NodeFactory.AddNodeAsPrototype('Vision/Basic Container Operations/F_VN_FillContainerExp/F_VN_FillContainerExp_DINT', node_F_VN_FillContainerExp_DINT);
NodeFactory.AddNodeAsPrototype('Vision/Basic Container Operations/F_VN_FillContainerExp/F_VN_FillContainerExp_INT', node_F_VN_FillContainerExp_INT);
NodeFactory.AddNodeAsPrototype('Vision/Basic Container Operations/F_VN_FillContainerExp/F_VN_FillContainerExp_ITcVnImage', node_F_VN_FillContainerExp_ITcVnImage);
NodeFactory.AddNodeAsPrototype('Vision/Basic Container Operations/F_VN_FillContainerExp/F_VN_FillContainerExp_LREAL', node_F_VN_FillContainerExp_LREAL);
NodeFactory.AddNodeAsPrototype('Vision/Basic Container Operations/F_VN_FillContainerExp/F_VN_FillContainerExp_REAL', node_F_VN_FillContainerExp_REAL);
NodeFactory.AddNodeAsPrototype('Vision/Basic Container Operations/F_VN_FillContainerExp/F_VN_FillContainerExp_SINT', node_F_VN_FillContainerExp_SINT);
NodeFactory.AddNodeAsPrototype('Vision/Basic Container Operations/F_VN_FillContainerExp/F_VN_FillContainerExp_TcVnDMatch', node_F_VN_FillContainerExp_TcVnDMatch);
NodeFactory.AddNodeAsPrototype('Vision/Basic Container Operations/F_VN_FillContainerExp/F_VN_FillContainerExp_TcVnKeyPoint', node_F_VN_FillContainerExp_TcVnKeyPoint);
NodeFactory.AddNodeAsPrototype('Vision/Basic Container Operations/F_VN_FillContainerExp/F_VN_FillContainerExp_TcVnPoint2_DINT', node_F_VN_FillContainerExp_TcVnPoint2_DINT);
NodeFactory.AddNodeAsPrototype('Vision/Basic Container Operations/F_VN_FillContainerExp/F_VN_FillContainerExp_TcVnPoint2_LREAL', node_F_VN_FillContainerExp_TcVnPoint2_LREAL);
NodeFactory.AddNodeAsPrototype('Vision/Basic Container Operations/F_VN_FillContainerExp/F_VN_FillContainerExp_TcVnPoint2_REAL', node_F_VN_FillContainerExp_TcVnPoint2_REAL);
NodeFactory.AddNodeAsPrototype('Vision/Basic Container Operations/F_VN_FillContainerExp/F_VN_FillContainerExp_TcVnPoint3_LREAL', node_F_VN_FillContainerExp_TcVnPoint3_LREAL);
NodeFactory.AddNodeAsPrototype('Vision/Basic Container Operations/F_VN_FillContainerExp/F_VN_FillContainerExp_TcVnPoint3_REAL', node_F_VN_FillContainerExp_TcVnPoint3_REAL);
NodeFactory.AddNodeAsPrototype('Vision/Basic Container Operations/F_VN_FillContainerExp/F_VN_FillContainerExp_TcVnRectangle_DINT', node_F_VN_FillContainerExp_TcVnRectangle_DINT);
NodeFactory.AddNodeAsPrototype('Vision/Basic Container Operations/F_VN_FillContainerExp/F_VN_FillContainerExp_TcVnRotatedRectangle', node_F_VN_FillContainerExp_TcVnRotatedRectangle);
NodeFactory.AddNodeAsPrototype('Vision/Basic Container Operations/F_VN_FillContainerExp/F_VN_FillContainerExp_TcVnVector2_DINT', node_F_VN_FillContainerExp_TcVnVector2_DINT);
NodeFactory.AddNodeAsPrototype('Vision/Basic Container Operations/F_VN_FillContainerExp/F_VN_FillContainerExp_TcVnVector2_INT', node_F_VN_FillContainerExp_TcVnVector2_INT);
NodeFactory.AddNodeAsPrototype('Vision/Basic Container Operations/F_VN_FillContainerExp/F_VN_FillContainerExp_TcVnVector2_REAL', node_F_VN_FillContainerExp_TcVnVector2_REAL);
NodeFactory.AddNodeAsPrototype('Vision/Basic Container Operations/F_VN_FillContainerExp/F_VN_FillContainerExp_TcVnVector2_SINT', node_F_VN_FillContainerExp_TcVnVector2_SINT);
NodeFactory.AddNodeAsPrototype('Vision/Basic Container Operations/F_VN_FillContainerExp/F_VN_FillContainerExp_TcVnVector2_UINT', node_F_VN_FillContainerExp_TcVnVector2_UINT);
NodeFactory.AddNodeAsPrototype('Vision/Basic Container Operations/F_VN_FillContainerExp/F_VN_FillContainerExp_TcVnVector2_USINT', node_F_VN_FillContainerExp_TcVnVector2_USINT);
NodeFactory.AddNodeAsPrototype('Vision/Basic Container Operations/F_VN_FillContainerExp/F_VN_FillContainerExp_TcVnVector3_INT', node_F_VN_FillContainerExp_TcVnVector3_INT);
NodeFactory.AddNodeAsPrototype('Vision/Basic Container Operations/F_VN_FillContainerExp/F_VN_FillContainerExp_TcVnVector3_REAL', node_F_VN_FillContainerExp_TcVnVector3_REAL);
NodeFactory.AddNodeAsPrototype('Vision/Basic Container Operations/F_VN_FillContainerExp/F_VN_FillContainerExp_TcVnVector3_SINT', node_F_VN_FillContainerExp_TcVnVector3_SINT);
NodeFactory.AddNodeAsPrototype('Vision/Basic Container Operations/F_VN_FillContainerExp/F_VN_FillContainerExp_TcVnVector3_UINT', node_F_VN_FillContainerExp_TcVnVector3_UINT);
NodeFactory.AddNodeAsPrototype('Vision/Basic Container Operations/F_VN_FillContainerExp/F_VN_FillContainerExp_TcVnVector3_USINT', node_F_VN_FillContainerExp_TcVnVector3_USINT);
NodeFactory.AddNodeAsPrototype('Vision/Basic Container Operations/F_VN_FillContainerExp/F_VN_FillContainerExp_TcVnVector4_DINT', node_F_VN_FillContainerExp_TcVnVector4_DINT);
NodeFactory.AddNodeAsPrototype('Vision/Basic Container Operations/F_VN_FillContainerExp/F_VN_FillContainerExp_TcVnVector4_INT', node_F_VN_FillContainerExp_TcVnVector4_INT);
NodeFactory.AddNodeAsPrototype('Vision/Basic Container Operations/F_VN_FillContainerExp/F_VN_FillContainerExp_TcVnVector4_LREAL', node_F_VN_FillContainerExp_TcVnVector4_LREAL);
NodeFactory.AddNodeAsPrototype('Vision/Basic Container Operations/F_VN_FillContainerExp/F_VN_FillContainerExp_TcVnVector4_REAL', node_F_VN_FillContainerExp_TcVnVector4_REAL);
NodeFactory.AddNodeAsPrototype('Vision/Basic Container Operations/F_VN_FillContainerExp/F_VN_FillContainerExp_TcVnVector4_SINT', node_F_VN_FillContainerExp_TcVnVector4_SINT);
NodeFactory.AddNodeAsPrototype('Vision/Basic Container Operations/F_VN_FillContainerExp/F_VN_FillContainerExp_TcVnVector4_UINT', node_F_VN_FillContainerExp_TcVnVector4_UINT);
NodeFactory.AddNodeAsPrototype('Vision/Basic Container Operations/F_VN_FillContainerExp/F_VN_FillContainerExp_TcVnVector4_USINT', node_F_VN_FillContainerExp_TcVnVector4_USINT);
NodeFactory.AddNodeAsPrototype('Vision/Basic Container Operations/F_VN_FillContainerExp/F_VN_FillContainerExp_UDINT', node_F_VN_FillContainerExp_UDINT);
NodeFactory.AddNodeAsPrototype('Vision/Basic Container Operations/F_VN_FillContainerExp/F_VN_FillContainerExp_UINT', node_F_VN_FillContainerExp_UINT);
NodeFactory.AddNodeAsPrototype('Vision/Basic Container Operations/F_VN_FillContainerExp/F_VN_FillContainerExp_ULINT', node_F_VN_FillContainerExp_ULINT);
NodeFactory.AddNodeAsPrototype('Vision/Basic Container Operations/F_VN_FillContainerExp/F_VN_FillContainerExp_USINT', node_F_VN_FillContainerExp_USINT);

NodeFactory.AddNodeAsPrototype('Vision/Basic Container Operations/F_VN_GetAt/F_VN_GetAt_DINT', node_F_VN_GetAt_DINT);
NodeFactory.AddNodeAsPrototype('Vision/Basic Container Operations/F_VN_GetAt/F_VN_GetAt_INT', node_F_VN_GetAt_INT);
NodeFactory.AddNodeAsPrototype('Vision/Basic Container Operations/F_VN_GetAt/F_VN_GetAt_ITcVnContainer', node_F_VN_GetAt_ITcVnContainer);
NodeFactory.AddNodeAsPrototype('Vision/Basic Container Operations/F_VN_GetAt/F_VN_GetAt_ITcVnImage', node_F_VN_GetAt_ITcVnImage);
NodeFactory.AddNodeAsPrototype('Vision/Basic Container Operations/F_VN_GetAt/F_VN_GetAt_LREAL', node_F_VN_GetAt_LREAL);
NodeFactory.AddNodeAsPrototype('Vision/Basic Container Operations/F_VN_GetAt/F_VN_GetAt_REAL', node_F_VN_GetAt_REAL);
NodeFactory.AddNodeAsPrototype('Vision/Basic Container Operations/F_VN_GetAt/F_VN_GetAt_SINT', node_F_VN_GetAt_SINT);
NodeFactory.AddNodeAsPrototype('Vision/Basic Container Operations/F_VN_GetAt/F_VN_GetAt_TcVnDMatch', node_F_VN_GetAt_TcVnDMatch);
NodeFactory.AddNodeAsPrototype('Vision/Basic Container Operations/F_VN_GetAt/F_VN_GetAt_TcVnKeyPoint', node_F_VN_GetAt_TcVnKeyPoint);
NodeFactory.AddNodeAsPrototype('Vision/Basic Container Operations/F_VN_GetAt/F_VN_GetAt_TcVnPoint2_DINT', node_F_VN_GetAt_TcVnPoint2_DINT);
NodeFactory.AddNodeAsPrototype('Vision/Basic Container Operations/F_VN_GetAt/F_VN_GetAt_TcVnPoint2_LREAL', node_F_VN_GetAt_TcVnPoint2_LREAL);
NodeFactory.AddNodeAsPrototype('Vision/Basic Container Operations/F_VN_GetAt/F_VN_GetAt_TcVnPoint2_REAL', node_F_VN_GetAt_TcVnPoint2_REAL);
NodeFactory.AddNodeAsPrototype('Vision/Basic Container Operations/F_VN_GetAt/F_VN_GetAt_TcVnPoint3_LREAL', node_F_VN_GetAt_TcVnPoint3_LREAL);
NodeFactory.AddNodeAsPrototype('Vision/Basic Container Operations/F_VN_GetAt/F_VN_GetAt_TcVnPoint3_REAL', node_F_VN_GetAt_TcVnPoint3_REAL);
NodeFactory.AddNodeAsPrototype('Vision/Basic Container Operations/F_VN_GetAt/F_VN_GetAt_TcVnRectangle_DINT', node_F_VN_GetAt_TcVnRectangle_DINT);
NodeFactory.AddNodeAsPrototype('Vision/Basic Container Operations/F_VN_GetAt/F_VN_GetAt_TcVnRotatedRectangle', node_F_VN_GetAt_TcVnRotatedRectangle);
NodeFactory.AddNodeAsPrototype('Vision/Basic Container Operations/F_VN_GetAt/F_VN_GetAt_TcVnVector2_DINT', node_F_VN_GetAt_TcVnVector2_DINT);
NodeFactory.AddNodeAsPrototype('Vision/Basic Container Operations/F_VN_GetAt/F_VN_GetAt_TcVnVector2_INT', node_F_VN_GetAt_TcVnVector2_INT);
NodeFactory.AddNodeAsPrototype('Vision/Basic Container Operations/F_VN_GetAt/F_VN_GetAt_TcVnVector2_REAL', node_F_VN_GetAt_TcVnVector2_REAL);
NodeFactory.AddNodeAsPrototype('Vision/Basic Container Operations/F_VN_GetAt/F_VN_GetAt_TcVnVector2_SINT', node_F_VN_GetAt_TcVnVector2_SINT);
NodeFactory.AddNodeAsPrototype('Vision/Basic Container Operations/F_VN_GetAt/F_VN_GetAt_TcVnVector2_UINT', node_F_VN_GetAt_TcVnVector2_UINT);
NodeFactory.AddNodeAsPrototype('Vision/Basic Container Operations/F_VN_GetAt/F_VN_GetAt_TcVnVector2_USINT', node_F_VN_GetAt_TcVnVector2_USINT);
NodeFactory.AddNodeAsPrototype('Vision/Basic Container Operations/F_VN_GetAt/F_VN_GetAt_TcVnVector3_INT', node_F_VN_GetAt_TcVnVector3_INT);
NodeFactory.AddNodeAsPrototype('Vision/Basic Container Operations/F_VN_GetAt/F_VN_GetAt_TcVnVector3_REAL', node_F_VN_GetAt_TcVnVector3_REAL);
NodeFactory.AddNodeAsPrototype('Vision/Basic Container Operations/F_VN_GetAt/F_VN_GetAt_TcVnVector3_SINT', node_F_VN_GetAt_TcVnVector3_SINT);
NodeFactory.AddNodeAsPrototype('Vision/Basic Container Operations/F_VN_GetAt/F_VN_GetAt_TcVnVector3_UINT', node_F_VN_GetAt_TcVnVector3_UINT);
NodeFactory.AddNodeAsPrototype('Vision/Basic Container Operations/F_VN_GetAt/F_VN_GetAt_TcVnVector3_USINT', node_F_VN_GetAt_TcVnVector3_USINT);
NodeFactory.AddNodeAsPrototype('Vision/Basic Container Operations/F_VN_GetAt/F_VN_GetAt_TcVnVector4_DINT', node_F_VN_GetAt_TcVnVector4_DINT);
NodeFactory.AddNodeAsPrototype('Vision/Basic Container Operations/F_VN_GetAt/F_VN_GetAt_TcVnVector4_INT', node_F_VN_GetAt_TcVnVector4_INT);
NodeFactory.AddNodeAsPrototype('Vision/Basic Container Operations/F_VN_GetAt/F_VN_GetAt_TcVnVector4_LREAL', node_F_VN_GetAt_TcVnVector4_LREAL);
NodeFactory.AddNodeAsPrototype('Vision/Basic Container Operations/F_VN_GetAt/F_VN_GetAt_TcVnVector4_REAL', node_F_VN_GetAt_TcVnVector4_REAL);
NodeFactory.AddNodeAsPrototype('Vision/Basic Container Operations/F_VN_GetAt/F_VN_GetAt_TcVnVector4_SINT', node_F_VN_GetAt_TcVnVector4_SINT);
NodeFactory.AddNodeAsPrototype('Vision/Basic Container Operations/F_VN_GetAt/F_VN_GetAt_TcVnVector4_UINT', node_F_VN_GetAt_TcVnVector4_UINT);
NodeFactory.AddNodeAsPrototype('Vision/Basic Container Operations/F_VN_GetAt/F_VN_GetAt_TcVnVector4_USINT', node_F_VN_GetAt_TcVnVector4_USINT);
NodeFactory.AddNodeAsPrototype('Vision/Basic Container Operations/F_VN_GetAt/F_VN_GetAt_UDINT', node_F_VN_GetAt_UDINT);
NodeFactory.AddNodeAsPrototype('Vision/Basic Container Operations/F_VN_GetAt/F_VN_GetAt_UINT', node_F_VN_GetAt_UINT);
NodeFactory.AddNodeAsPrototype('Vision/Basic Container Operations/F_VN_GetAt/F_VN_GetAt_ULINT', node_F_VN_GetAt_ULINT);
NodeFactory.AddNodeAsPrototype('Vision/Basic Container Operations/F_VN_GetAt/F_VN_GetAt_USINT', node_F_VN_GetAt_USINT);

NodeFactory.AddNodeAsPrototype('Vision/Basic Container Operations/F_VN_InsertIntoContainer/F_VN_InsertIntoContainer_DINT', node_F_VN_InsertIntoContainer_DINT);
NodeFactory.AddNodeAsPrototype('Vision/Basic Container Operations/F_VN_InsertIntoContainer/F_VN_InsertIntoContainer_INT', node_F_VN_InsertIntoContainer_INT);
NodeFactory.AddNodeAsPrototype('Vision/Basic Container Operations/F_VN_InsertIntoContainer/F_VN_InsertIntoContainer_ITcVnContainer', node_F_VN_InsertIntoContainer_ITcVnContainer);
//NodeFactory.AddNodeAsPrototype('Vision/Basic Container Operations/F_VN_InsertIntoContainer/F_VN_InsertIntoContainer_ITcVnForwardIterator', node_F_VN_InsertIntoContainer_ITcVnForwardIterator);
NodeFactory.AddNodeAsPrototype('Vision/Basic Container Operations/F_VN_InsertIntoContainer/F_VN_InsertIntoContainer_ITcVnImage', node_F_VN_InsertIntoContainer_ITcVnImage);
NodeFactory.AddNodeAsPrototype('Vision/Basic Container Operations/F_VN_InsertIntoContainer/F_VN_InsertIntoContainer_LREAL', node_F_VN_InsertIntoContainer_LREAL);
NodeFactory.AddNodeAsPrototype('Vision/Basic Container Operations/F_VN_InsertIntoContainer/F_VN_InsertIntoContainer_REAL', node_F_VN_InsertIntoContainer_REAL);
NodeFactory.AddNodeAsPrototype('Vision/Basic Container Operations/F_VN_InsertIntoContainer/F_VN_InsertIntoContainer_SINT', node_F_VN_InsertIntoContainer_SINT);
NodeFactory.AddNodeAsPrototype('Vision/Basic Container Operations/F_VN_InsertIntoContainer/F_VN_InsertIntoContainer_TcVnDMatch', node_F_VN_InsertIntoContainer_TcVnDMatch);
NodeFactory.AddNodeAsPrototype('Vision/Basic Container Operations/F_VN_InsertIntoContainer/F_VN_InsertIntoContainer_TcVnKeyPoint', node_F_VN_InsertIntoContainer_TcVnKeyPoint);
NodeFactory.AddNodeAsPrototype('Vision/Basic Container Operations/F_VN_InsertIntoContainer/F_VN_InsertIntoContainer_TcVnPoint2_DINT', node_F_VN_InsertIntoContainer_TcVnPoint2_DINT);
NodeFactory.AddNodeAsPrototype('Vision/Basic Container Operations/F_VN_InsertIntoContainer/F_VN_InsertIntoContainer_TcVnPoint2_LREAL', node_F_VN_InsertIntoContainer_TcVnPoint2_LREAL);
NodeFactory.AddNodeAsPrototype('Vision/Basic Container Operations/F_VN_InsertIntoContainer/F_VN_InsertIntoContainer_TcVnPoint2_REAL', node_F_VN_InsertIntoContainer_TcVnPoint2_REAL);
NodeFactory.AddNodeAsPrototype('Vision/Basic Container Operations/F_VN_InsertIntoContainer/F_VN_InsertIntoContainer_TcVnPoint3_LREAL', node_F_VN_InsertIntoContainer_TcVnPoint3_LREAL);
NodeFactory.AddNodeAsPrototype('Vision/Basic Container Operations/F_VN_InsertIntoContainer/F_VN_InsertIntoContainer_TcVnPoint3_REAL', node_F_VN_InsertIntoContainer_TcVnPoint3_REAL);
NodeFactory.AddNodeAsPrototype('Vision/Basic Container Operations/F_VN_InsertIntoContainer/F_VN_InsertIntoContainer_TcVnRectangle_DINT', node_F_VN_InsertIntoContainer_TcVnRectangle_DINT);
NodeFactory.AddNodeAsPrototype('Vision/Basic Container Operations/F_VN_InsertIntoContainer/F_VN_InsertIntoContainer_TcVnRotatedRectangle', node_F_VN_InsertIntoContainer_TcVnRotatedRectangle);
NodeFactory.AddNodeAsPrototype('Vision/Basic Container Operations/F_VN_InsertIntoContainer/F_VN_InsertIntoContainer_TcVnVector2_DINT', node_F_VN_InsertIntoContainer_TcVnVector2_DINT);
NodeFactory.AddNodeAsPrototype('Vision/Basic Container Operations/F_VN_InsertIntoContainer/F_VN_InsertIntoContainer_TcVnVector2_INT', node_F_VN_InsertIntoContainer_TcVnVector2_INT);
NodeFactory.AddNodeAsPrototype('Vision/Basic Container Operations/F_VN_InsertIntoContainer/F_VN_InsertIntoContainer_TcVnVector2_REAL', node_F_VN_InsertIntoContainer_TcVnVector2_REAL);
NodeFactory.AddNodeAsPrototype('Vision/Basic Container Operations/F_VN_InsertIntoContainer/F_VN_InsertIntoContainer_TcVnVector2_SINT', node_F_VN_InsertIntoContainer_TcVnVector2_SINT);
NodeFactory.AddNodeAsPrototype('Vision/Basic Container Operations/F_VN_InsertIntoContainer/F_VN_InsertIntoContainer_TcVnVector2_UINT', node_F_VN_InsertIntoContainer_TcVnVector2_UINT);
NodeFactory.AddNodeAsPrototype('Vision/Basic Container Operations/F_VN_InsertIntoContainer/F_VN_InsertIntoContainer_TcVnVector2_USINT', node_F_VN_InsertIntoContainer_TcVnVector2_USINT);
NodeFactory.AddNodeAsPrototype('Vision/Basic Container Operations/F_VN_InsertIntoContainer/F_VN_InsertIntoContainer_TcVnVector3_INT', node_F_VN_InsertIntoContainer_TcVnVector3_INT);
NodeFactory.AddNodeAsPrototype('Vision/Basic Container Operations/F_VN_InsertIntoContainer/F_VN_InsertIntoContainer_TcVnVector3_REAL', node_F_VN_InsertIntoContainer_TcVnVector3_REAL);
NodeFactory.AddNodeAsPrototype('Vision/Basic Container Operations/F_VN_InsertIntoContainer/F_VN_InsertIntoContainer_TcVnVector3_SINT', node_F_VN_InsertIntoContainer_TcVnVector3_SINT);
NodeFactory.AddNodeAsPrototype('Vision/Basic Container Operations/F_VN_InsertIntoContainer/F_VN_InsertIntoContainer_TcVnVector3_UINT', node_F_VN_InsertIntoContainer_TcVnVector3_UINT);
NodeFactory.AddNodeAsPrototype('Vision/Basic Container Operations/F_VN_InsertIntoContainer/F_VN_InsertIntoContainer_TcVnVector3_USINT', node_F_VN_InsertIntoContainer_TcVnVector3_USINT);
NodeFactory.AddNodeAsPrototype('Vision/Basic Container Operations/F_VN_InsertIntoContainer/F_VN_InsertIntoContainer_TcVnVector4_DINT', node_F_VN_InsertIntoContainer_TcVnVector4_DINT);
NodeFactory.AddNodeAsPrototype('Vision/Basic Container Operations/F_VN_InsertIntoContainer/F_VN_InsertIntoContainer_TcVnVector4_INT', node_F_VN_InsertIntoContainer_TcVnVector4_INT);
NodeFactory.AddNodeAsPrototype('Vision/Basic Container Operations/F_VN_InsertIntoContainer/F_VN_InsertIntoContainer_TcVnVector4_LREAL', node_F_VN_InsertIntoContainer_TcVnVector4_LREAL);
NodeFactory.AddNodeAsPrototype('Vision/Basic Container Operations/F_VN_InsertIntoContainer/F_VN_InsertIntoContainer_TcVnVector4_REAL', node_F_VN_InsertIntoContainer_TcVnVector4_REAL);
NodeFactory.AddNodeAsPrototype('Vision/Basic Container Operations/F_VN_InsertIntoContainer/F_VN_InsertIntoContainer_TcVnVector4_SINT', node_F_VN_InsertIntoContainer_TcVnVector4_SINT);
NodeFactory.AddNodeAsPrototype('Vision/Basic Container Operations/F_VN_InsertIntoContainer/F_VN_InsertIntoContainer_TcVnVector4_UINT', node_F_VN_InsertIntoContainer_TcVnVector4_UINT);
NodeFactory.AddNodeAsPrototype('Vision/Basic Container Operations/F_VN_InsertIntoContainer/F_VN_InsertIntoContainer_TcVnVector4_USINT', node_F_VN_InsertIntoContainer_TcVnVector4_USINT);
NodeFactory.AddNodeAsPrototype('Vision/Basic Container Operations/F_VN_InsertIntoContainer/F_VN_InsertIntoContainer_UDINT', node_F_VN_InsertIntoContainer_UDINT);
NodeFactory.AddNodeAsPrototype('Vision/Basic Container Operations/F_VN_InsertIntoContainer/F_VN_InsertIntoContainer_UINT', node_F_VN_InsertIntoContainer_UINT);
NodeFactory.AddNodeAsPrototype('Vision/Basic Container Operations/F_VN_InsertIntoContainer/F_VN_InsertIntoContainer_ULINT', node_F_VN_InsertIntoContainer_ULINT);
NodeFactory.AddNodeAsPrototype('Vision/Basic Container Operations/F_VN_InsertIntoContainer/F_VN_InsertIntoContainer_USINT', node_F_VN_InsertIntoContainer_USINT);

NodeFactory.AddNodeAsPrototype('Vision/Basic Container Operations/F_VN_SetAt/F_VN_SetAt_DINT', node_F_VN_SetAt_DINT);
NodeFactory.AddNodeAsPrototype('Vision/Basic Container Operations/F_VN_SetAt/F_VN_SetAt_INT', node_F_VN_SetAt_INT);
NodeFactory.AddNodeAsPrototype('Vision/Basic Container Operations/F_VN_SetAt/F_VN_SetAt_ITcVnContainer', node_F_VN_SetAt_ITcVnContainer);
NodeFactory.AddNodeAsPrototype('Vision/Basic Container Operations/F_VN_SetAt/F_VN_SetAt_ITcVnImage', node_F_VN_SetAt_ITcVnImage);
NodeFactory.AddNodeAsPrototype('Vision/Basic Container Operations/F_VN_SetAt/F_VN_SetAt_LREAL', node_F_VN_SetAt_LREAL);
NodeFactory.AddNodeAsPrototype('Vision/Basic Container Operations/F_VN_SetAt/F_VN_SetAt_REAL', node_F_VN_SetAt_REAL);
NodeFactory.AddNodeAsPrototype('Vision/Basic Container Operations/F_VN_SetAt/F_VN_SetAt_SINT', node_F_VN_SetAt_SINT);
NodeFactory.AddNodeAsPrototype('Vision/Basic Container Operations/F_VN_SetAt/F_VN_SetAt_TcVnDMatch', node_F_VN_SetAt_TcVnDMatch);
NodeFactory.AddNodeAsPrototype('Vision/Basic Container Operations/F_VN_SetAt/F_VN_SetAt_TcVnKeyPoint', node_F_VN_SetAt_TcVnKeyPoint);
NodeFactory.AddNodeAsPrototype('Vision/Basic Container Operations/F_VN_SetAt/F_VN_SetAt_TcVnPoint2_DINT', node_F_VN_SetAt_TcVnPoint2_DINT);
NodeFactory.AddNodeAsPrototype('Vision/Basic Container Operations/F_VN_SetAt/F_VN_SetAt_TcVnPoint2_LREAL', node_F_VN_SetAt_TcVnPoint2_LREAL);
NodeFactory.AddNodeAsPrototype('Vision/Basic Container Operations/F_VN_SetAt/F_VN_SetAt_TcVnPoint2_REAL', node_F_VN_SetAt_TcVnPoint2_REAL);
NodeFactory.AddNodeAsPrototype('Vision/Basic Container Operations/F_VN_SetAt/F_VN_SetAt_TcVnPoint3_LREAL', node_F_VN_SetAt_TcVnPoint3_LREAL);
NodeFactory.AddNodeAsPrototype('Vision/Basic Container Operations/F_VN_SetAt/F_VN_SetAt_TcVnPoint3_REAL', node_F_VN_SetAt_TcVnPoint3_REAL);
NodeFactory.AddNodeAsPrototype('Vision/Basic Container Operations/F_VN_SetAt/F_VN_SetAt_TcVnRectangle_DINT', node_F_VN_SetAt_TcVnRectangle_DINT);
NodeFactory.AddNodeAsPrototype('Vision/Basic Container Operations/F_VN_SetAt/F_VN_SetAt_TcVnRotatedRectangle', node_F_VN_SetAt_TcVnRotatedRectangle);
NodeFactory.AddNodeAsPrototype('Vision/Basic Container Operations/F_VN_SetAt/F_VN_SetAt_TcVnVector2_DINT', node_F_VN_SetAt_TcVnVector2_DINT);
NodeFactory.AddNodeAsPrototype('Vision/Basic Container Operations/F_VN_SetAt/F_VN_SetAt_TcVnVector2_INT', node_F_VN_SetAt_TcVnVector2_INT);
NodeFactory.AddNodeAsPrototype('Vision/Basic Container Operations/F_VN_SetAt/F_VN_SetAt_TcVnVector2_REAL', node_F_VN_SetAt_TcVnVector2_REAL);
NodeFactory.AddNodeAsPrototype('Vision/Basic Container Operations/F_VN_SetAt/F_VN_SetAt_TcVnVector2_SINT', node_F_VN_SetAt_TcVnVector2_SINT);
NodeFactory.AddNodeAsPrototype('Vision/Basic Container Operations/F_VN_SetAt/F_VN_SetAt_TcVnVector2_UINT', node_F_VN_SetAt_TcVnVector2_UINT);
NodeFactory.AddNodeAsPrototype('Vision/Basic Container Operations/F_VN_SetAt/F_VN_SetAt_TcVnVector2_USINT', node_F_VN_SetAt_TcVnVector2_USINT);
NodeFactory.AddNodeAsPrototype('Vision/Basic Container Operations/F_VN_SetAt/F_VN_SetAt_TcVnVector3_INT', node_F_VN_SetAt_TcVnVector3_INT);
NodeFactory.AddNodeAsPrototype('Vision/Basic Container Operations/F_VN_SetAt/F_VN_SetAt_TcVnVector3_REAL', node_F_VN_SetAt_TcVnVector3_REAL);
NodeFactory.AddNodeAsPrototype('Vision/Basic Container Operations/F_VN_SetAt/F_VN_SetAt_TcVnVector3_SINT', node_F_VN_SetAt_TcVnVector3_SINT);
NodeFactory.AddNodeAsPrototype('Vision/Basic Container Operations/F_VN_SetAt/F_VN_SetAt_TcVnVector3_UINT', node_F_VN_SetAt_TcVnVector3_UINT);
NodeFactory.AddNodeAsPrototype('Vision/Basic Container Operations/F_VN_SetAt/F_VN_SetAt_TcVnVector3_USINT', node_F_VN_SetAt_TcVnVector3_USINT);
NodeFactory.AddNodeAsPrototype('Vision/Basic Container Operations/F_VN_SetAt/F_VN_SetAt_TcVnVector4_DINT', node_F_VN_SetAt_TcVnVector4_DINT);
NodeFactory.AddNodeAsPrototype('Vision/Basic Container Operations/F_VN_SetAt/F_VN_SetAt_TcVnVector4_INT', node_F_VN_SetAt_TcVnVector4_INT);
NodeFactory.AddNodeAsPrototype('Vision/Basic Container Operations/F_VN_SetAt/F_VN_SetAt_TcVnVector4_LREAL', node_F_VN_SetAt_TcVnVector4_LREAL);
NodeFactory.AddNodeAsPrototype('Vision/Basic Container Operations/F_VN_SetAt/F_VN_SetAt_TcVnVector4_REAL', node_F_VN_SetAt_TcVnVector4_REAL);
NodeFactory.AddNodeAsPrototype('Vision/Basic Container Operations/F_VN_SetAt/F_VN_SetAt_TcVnVector4_SINT', node_F_VN_SetAt_TcVnVector4_SINT);
NodeFactory.AddNodeAsPrototype('Vision/Basic Container Operations/F_VN_SetAt/F_VN_SetAt_TcVnVector4_UINT', node_F_VN_SetAt_TcVnVector4_UINT);
NodeFactory.AddNodeAsPrototype('Vision/Basic Container Operations/F_VN_SetAt/F_VN_SetAt_TcVnVector4_USINT', node_F_VN_SetAt_TcVnVector4_USINT);
NodeFactory.AddNodeAsPrototype('Vision/Basic Container Operations/F_VN_SetAt/F_VN_SetAt_UDINT', node_F_VN_SetAt_UDINT);
NodeFactory.AddNodeAsPrototype('Vision/Basic Container Operations/F_VN_SetAt/F_VN_SetAt_UINT', node_F_VN_SetAt_UINT);
NodeFactory.AddNodeAsPrototype('Vision/Basic Container Operations/F_VN_SetAt/F_VN_SetAt_ULINT', node_F_VN_SetAt_ULINT);
NodeFactory.AddNodeAsPrototype('Vision/Basic Container Operations/F_VN_SetAt/F_VN_SetAt_USINT', node_F_VN_SetAt_USINT);

//NodeFactory.AddNodeAsPrototype('Vision/Basic Container Operations/F_VN_AdvanceIterator', node_F_VN_AdvanceIterator);
NodeFactory.AddNodeAsPrototype('Vision/Basic Container Operations/F_VN_CheckIfEmpty', node_F_VN_CheckIfEmpty);
//NodeFactory.AddNodeAsPrototype('Vision/Basic Container Operations/F_VN_CheckIfIteratorIsAtEnd', node_F_VN_CheckIfIteratorIsAtEnd);
//NodeFactory.AddNodeAsPrototype('Vision/Basic Container Operations/F_VN_ConvertContainerType', node_F_VN_ConvertContainerType);
NodeFactory.AddNodeAsPrototype('Vision/Basic Container Operations/F_VN_CopyContainer', node_F_VN_CopyContainer);
//NodeFactory.AddNodeAsPrototype('Vision/Basic Container Operations/F_VN_CopyContainerElementsConditional_ITcVnContainer', node_F_VN_CopyContainerElementsConditional_ITcVnContainer);
//NodeFactory.AddNodeAsPrototype('Vision/Basic Container Operations/F_VN_CopyContainerElementsConditional_ITcVnForwardIterator', node_F_VN_CopyContainerElementsConditional_ITcVnForwardIterator);
NodeFactory.AddNodeAsPrototype('Vision/Basic Container Operations/F_VN_CreateContainer', node_F_VN_CreateContainer);
//NodeFactory.AddNodeAsPrototype('Vision/Basic Container Operations/F_VN_CreateContainerFromArray', node_F_VN_CreateContainerFromArray);
//NodeFactory.AddNodeAsPrototype('Vision/Basic Container Operations/F_VN_EraseFromContainer', node_F_VN_EraseFromContainer);
//NodeFactory.AddNodeAsPrototype('Vision/Basic Container Operations/F_VN_ExportContainer', node_F_VN_ExportContainer);
NodeFactory.AddNodeAsPrototype('Vision/Basic Container Operations/F_VN_ExportContainer_String', node_F_VN_ExportContainer_String);
//NodeFactory.AddNodeAsPrototype('Vision/Basic Container Operations/F_VN_ExportContainerSize', node_F_VN_ExportContainerSize);
//NodeFactory.AddNodeAsPrototype('Vision/Basic Container Operations/F_VN_ExportSubContainer', node_F_VN_ExportSubContainer);
NodeFactory.AddNodeAsPrototype('Vision/Basic Container Operations/F_VN_ExportSubContainer_String', node_F_VN_ExportSubContainer_String);
//NodeFactory.AddNodeAsPrototype('Vision/Basic Container Operations/F_VN_ExportSubContainerSize', node_F_VN_ExportSubContainerSize);
NodeFactory.AddNodeAsPrototype('Vision/Basic Container Operations/F_VN_ExtractContainerRange', node_F_VN_ExtractContainerRange);
//NodeFactory.AddNodeAsPrototype('Vision/Basic Container Operations/F_VN_GetContainer', node_F_VN_GetContainer);
//NodeFactory.AddNodeAsPrototype('Vision/Basic Container Operations/F_VN_GetContainerExp', node_F_VN_GetContainerExp);
//NodeFactory.AddNodeAsPrototype('Vision/Basic Container Operations/F_VN_GetForwardIterator', node_F_VN_GetForwardIterator);
NodeFactory.AddNodeAsPrototype('Vision/Basic Container Operations/F_VN_GetNumberOfElements', node_F_VN_GetNumberOfElements);
//NodeFactory.AddNodeAsPrototype('Vision/Basic Container Operations/F_VN_GetRandomAccessIterator', node_F_VN_GetRandomAccessIterator);
//NodeFactory.AddNodeAsPrototype('Vision/Basic Container Operations/F_VN_IncrementIterator', node_F_VN_IncrementIterator);
//NodeFactory.AddNodeAsPrototype('Vision/Basic Container Operations/F_VN_IteratorDistance', node_F_VN_IteratorDistance);
//NodeFactory.AddNodeAsPrototype('Vision/Basic Container Operations/F_VN_ReserveContainerMemory', node_F_VN_ReserveContainerMemory);
NodeFactory.AddNodeAsPrototype('Vision/Basic Container Operations/F_VN_ReverseContainer', node_F_VN_ReverseContainer);
//NodeFactory.AddNodeAsPrototype('Vision/Basic Container Operations/F_VN_SetContainer', node_F_VN_SetContainer);
//NodeFactory.AddNodeAsPrototype('Vision/Basic Container Operations/F_VN_SetIteratorToBegin', node_F_VN_SetIteratorToBegin);

// Basic Image Operations
//NodeFactory.AddNodeAsPrototype('Vision/Basic Image Operations/F_VN_CombineImageChannels', node_F_VN_CombineImageChannels);
NodeFactory.AddNodeAsPrototype('Vision/Basic Image Operations/F_VN_ConvertElementType', node_F_VN_ConvertElementType);
NodeFactory.AddNodeAsPrototype('Vision/Basic Image Operations/F_VN_ConvertElementTypeExp', node_F_VN_ConvertElementTypeExp);
NodeFactory.AddNodeAsPrototype('Vision/Basic Image Operations/F_VN_CopyImage', node_F_VN_CopyImage);
NodeFactory.AddNodeAsPrototype('Vision/Basic Image Operations/F_VN_CopyImageRegion', node_F_VN_CopyImageRegion);
NodeFactory.AddNodeAsPrototype('Vision/Basic Image Operations/F_VN_CopyImageRegionToRegion', node_F_VN_CopyImageRegionToRegion);
NodeFactory.AddNodeAsPrototype('Vision/Basic Image Operations/F_VN_CopyIntoDisplayableImage', node_F_VN_CopyIntoDisplayableImage);
NodeFactory.AddNodeAsPrototype('Vision/Basic Image Operations/F_VN_CreateAssociatedImage', node_F_VN_CreateAssociatedImage);
NodeFactory.AddNodeAsPrototype('Vision/Basic Image Operations/F_VN_CreateEmptyImage', node_F_VN_CreateEmptyImage);
NodeFactory.AddNodeAsPrototype('Vision/Basic Image Operations/F_VN_CreateImage', node_F_VN_CreateImage);
NodeFactory.AddNodeAsPrototype('Vision/Basic Image Operations/F_VN_CreateImageAndSetPixels', node_F_VN_CreateImageAndSetPixels);
//NodeFactory.AddNodeAsPrototype('Vision/Basic Image Operations/F_VN_CreateImageFromArray', node_F_VN_CreateImageFromArray);
//NodeFactory.AddNodeAsPrototype('Vision/Basic Image Operations/F_VN_ExportImage', node_F_VN_ExportImage);
//NodeFactory.AddNodeAsPrototype('Vision/Basic Image Operations/F_VN_ExportImageAsBmp', node_F_VN_ExportImageAsBmp);
//NodeFactory.AddNodeAsPrototype('Vision/Basic Image Operations/F_VN_ExportImageAsBmpExp', node_F_VN_ExportImageAsBmpExp);
NodeFactory.AddNodeAsPrototype('Vision/Basic Image Operations/F_VN_ExportImageAsBmpSize', node_F_VN_ExportImageAsBmpSize);
NodeFactory.AddNodeAsPrototype('Vision/Basic Image Operations/F_VN_ExportImageAsBmpSizeExp', node_F_VN_ExportImageAsBmpSizeExp);
NodeFactory.AddNodeAsPrototype('Vision/Basic Image Operations/F_VN_ExportImageSize', node_F_VN_ExportImageSize);
NodeFactory.AddNodeAsPrototype('Vision/Basic Image Operations/F_VN_FuseImages', node_F_VN_FuseImages);
//NodeFactory.AddNodeAsPrototype('Vision/Basic Image Operations/F_VN_FuseImagesArray', node_F_VN_FuseImagesArray);
NodeFactory.AddNodeAsPrototype('Vision/Basic Image Operations/F_VN_GetImageChannel', node_F_VN_GetImageChannel);
NodeFactory.AddNodeAsPrototype('Vision/Basic Image Operations/F_VN_GetImageHeight', node_F_VN_GetImageHeight);
NodeFactory.AddNodeAsPrototype('Vision/Basic Image Operations/F_VN_GetImageInfo', node_F_VN_GetImageInfo);
NodeFactory.AddNodeAsPrototype('Vision/Basic Image Operations/F_VN_GetImageWidth', node_F_VN_GetImageWidth);
NodeFactory.AddNodeAsPrototype('Vision/Basic Image Operations/F_VN_GetPixel', node_F_VN_GetPixel);
NodeFactory.AddNodeAsPrototype('Vision/Basic Image Operations/F_VN_GetPixelFormat', node_F_VN_GetPixelFormat);
NodeFactory.AddNodeAsPrototype('Vision/Basic Image Operations/F_VN_GetRoi', node_F_VN_GetRoi);
NodeFactory.AddNodeAsPrototype('Vision/Basic Image Operations/F_VN_MixImageChannels', node_F_VN_MixImageChannels);
NodeFactory.AddNodeAsPrototype('Vision/Basic Image Operations/F_VN_ResetRoi', node_F_VN_ResetRoi);
NodeFactory.AddNodeAsPrototype('Vision/Basic Image Operations/F_VN_SetImageChannel', node_F_VN_SetImageChannel);
NodeFactory.AddNodeAsPrototype('Vision/Basic Image Operations/F_VN_SetPixel', node_F_VN_SetPixel);
NodeFactory.AddNodeAsPrototype('Vision/Basic Image Operations/F_VN_SetPixels', node_F_VN_SetPixels);
NodeFactory.AddNodeAsPrototype('Vision/Basic Image Operations/F_VN_SetPixelsExp', node_F_VN_SetPixelsExp);
NodeFactory.AddNodeAsPrototype('Vision/Basic Image Operations/F_VN_SetRoi', node_F_VN_SetRoi);
NodeFactory.AddNodeAsPrototype('Vision/Basic Image Operations/F_VN_SetRoi_TcVnRectangle_DINT', node_F_VN_SetRoi_TcVnRectangle_DINT);
NodeFactory.AddNodeAsPrototype('Vision/Basic Image Operations/F_VN_SetRoi_TcVnRectangle_UDINT', node_F_VN_SetRoi_TcVnRectangle_UDINT);
//NodeFactory.AddNodeAsPrototype('Vision/Basic Image Operations/F_VN_SplitImageChannels, node_F_VN_SplitImageChannels);
NodeFactory.AddNodeAsPrototype('Vision/Basic Image Operations/F_VN_TransformIntoDisplayableImage', node_F_VN_TransformIntoDisplayableImage); 
NodeFactory.AddNodeAsPrototype('Vision/Basic Image Operations/F_VN_TransformIntoDisplayableImageExp', node_F_VN_TransformIntoDisplayableImageExp); 
NodeFactory.AddNodeAsPrototype('Vision/Basic Image Operations/F_VN_CreateNDimensionalImage', node_F_VN_CreateNDimensionalImage);
NodeFactory.AddNodeAsPrototype('Vision/Basic Image Operations/F_VN_CreateNDimensionalImageAndSetPixels', node_F_VN_CreateNDimensionalImageAndSetPixels);
//NodeFactory.AddNodeAsPrototype('Vision/Basic Image Operations/F_VN_CreateNDimensionalImageFromArray, node_F_VN_CreateNDimensionalImageFromArray);
NodeFactory.AddNodeAsPrototype('Vision/Basic Image Operations/F_VN_GetLayoutInfo', node_F_VN_GetLayoutInfo);
NodeFactory.AddNodeAsPrototype('Vision/Basic Image Operations/F_VN_PadImageBorder', node_F_VN_PadImageBorder);
NodeFactory.AddNodeAsPrototype('Vision/Basic Image Operations/F_VN_PadImageBorderExp', node_F_VN_PadImageBorderExp);
//NodeFactory.AddNodeAsPrototype('Vision/Basic Image Operations/F_VN_ReinterpretUnsupportedImage', node_F_VN_ReinterpretUnsupportedImage);

// Code Quality
NodeFactory.AddNodeAsPrototype('Vision/Code Quality/F_VN_GradeBarcode', node_F_VN_GradeBarcode);
NodeFactory.AddNodeAsPrototype('Vision/Code Quality/F_VN_GradeBarcodeExp', node_F_VN_GradeBarcodeExp);
NodeFactory.AddNodeAsPrototype('Vision/Code Quality/F_VN_GradeDataMatrixCode', node_F_VN_GradeDataMatrixCode);
NodeFactory.AddNodeAsPrototype('Vision/Code Quality/F_VN_GradeDataMatrixCodeExp', node_F_VN_GradeDataMatrixCodeExp);
NodeFactory.AddNodeAsPrototype('Vision/Code Quality/F_VN_GradeQRCode', node_F_VN_GradeQRCode);
NodeFactory.AddNodeAsPrototype('Vision/Code Quality/F_VN_GradeQRCodeExp', node_F_VN_GradeQRCodeExp);

// Code Reading
NodeFactory.AddNodeAsPrototype('Vision/Code Reading/F_VN_AnalyzeBarcodeWalsh', node_F_VN_AnalyzeBarcodeWalsh);
NodeFactory.AddNodeAsPrototype('Vision/Code Reading/F_VN_DetectBarcodesWalsh', node_F_VN_DetectBarcodesWalsh);
NodeFactory.AddNodeAsPrototype('Vision/Code Reading/F_VN_DetectCodesNeuralNetwork', node_F_VN_DetectCodesNeuralNetwork);
NodeFactory.AddNodeAsPrototype('Vision/Code Reading/F_VN_ReadBarcode', node_F_VN_ReadBarcode);
NodeFactory.AddNodeAsPrototype('Vision/Code Reading/F_VN_ReadBarcodeExp', node_F_VN_ReadBarcodeExp);
NodeFactory.AddNodeAsPrototype('Vision/Code Reading/F_VN_ReadBarcodeExp2', node_F_VN_ReadBarcodeExp2);
NodeFactory.AddNodeAsPrototype('Vision/Code Reading/F_VN_ReadBarcodeRoi', node_F_VN_ReadBarcodeRoi);
NodeFactory.AddNodeAsPrototype('Vision/Code Reading/F_VN_ReadBarcodeRoiExp', node_F_VN_ReadBarcodeRoiExp);
NodeFactory.AddNodeAsPrototype('Vision/Code Reading/F_VN_ReadDataMatrixCode', node_F_VN_ReadDataMatrixCode);
NodeFactory.AddNodeAsPrototype('Vision/Code Reading/F_VN_ReadDataMatrixCodeExp', node_F_VN_ReadDataMatrixCodeExp);
NodeFactory.AddNodeAsPrototype('Vision/Code Reading/F_VN_ReadDataMatrixCodeExp2', node_F_VN_ReadDataMatrixCodeExp2);
NodeFactory.AddNodeAsPrototype('Vision/Code Reading/F_VN_ReadDataMatrixCodeRoi', node_F_VN_ReadDataMatrixCodeRoi);
NodeFactory.AddNodeAsPrototype('Vision/Code Reading/F_VN_ReadDataMatrixCodeRoiExp', node_F_VN_ReadDataMatrixCodeRoiExp);
NodeFactory.AddNodeAsPrototype('Vision/Code Reading/F_VN_ReadDotCodeRoi', Node_F_VN_ReadDotCodeRoi);
NodeFactory.AddNodeAsPrototype('Vision/Code Reading/F_VN_ReadDotCodeRoiExp', Node_F_VN_ReadDotCodeRoiExp);
NodeFactory.AddNodeAsPrototype('Vision/Code Reading/F_VN_ReadPharmaCode', node_F_VN_ReadPharmaCode);
NodeFactory.AddNodeAsPrototype('Vision/Code Reading/F_VN_ReadPharmaCodeExp', node_F_VN_ReadPharmaCodeExp);
NodeFactory.AddNodeAsPrototype('Vision/Code Reading/F_VN_ReadPharmaCodeExp2', node_F_VN_ReadPharmaCodeExp2);
NodeFactory.AddNodeAsPrototype('Vision/Code Reading/F_VN_ReadQRCode', node_F_VN_ReadQRCode);
NodeFactory.AddNodeAsPrototype('Vision/Code Reading/F_VN_ReadQRCodeExp', node_F_VN_ReadQRCodeExp);
NodeFactory.AddNodeAsPrototype('Vision/Code Reading/F_VN_ReadQRCodeExp2', node_F_VN_ReadQRCodeExp2);

// Constants
NodeFactory.AddNodeAsPrototype('Vision/Constants/RGBA_BLACK', node_RGBA_BLACK);
NodeFactory.AddNodeAsPrototype('Vision/Constants/RGBA_RED', node_RGBA_RED);
NodeFactory.AddNodeAsPrototype('Vision/Constants/RGBA_YELLOW', node_RGBA_YELLOW);
NodeFactory.AddNodeAsPrototype('Vision/Constants/RGBA_GREEN', node_RGBA_GREEN);
NodeFactory.AddNodeAsPrototype('Vision/Constants/RGBA_CYAN', node_RGBA_CYAN);
NodeFactory.AddNodeAsPrototype('Vision/Constants/RGBA_BLUE', node_RGBA_BLUE);
NodeFactory.AddNodeAsPrototype('Vision/Constants/RGBA_MAGENTA', node_RGBA_MAGENTA);
NodeFactory.AddNodeAsPrototype('Vision/Constants/RGBA_WHITE', node_RGBA_WHITE);
NodeFactory.AddNodeAsPrototype('Vision/Constants/RGBA_RANDOM', node_RGBA_RANDOM);
NodeFactory.AddNodeAsPrototype('Vision/Constants/ContainerType_Vector_SINT', node_ContainerType_Vector_SINT);
NodeFactory.AddNodeAsPrototype('Vision/Constants/ContainerType_Vector_USINT', node_ContainerType_Vector_USINT);
NodeFactory.AddNodeAsPrototype('Vision/Constants/ContainerType_Vector_INT', node_ContainerType_Vector_INT);
NodeFactory.AddNodeAsPrototype('Vision/Constants/ContainerType_Vector_UINT', node_ContainerType_Vector_UINT);
NodeFactory.AddNodeAsPrototype('Vision/Constants/ContainerType_Vector_DINT', node_ContainerType_Vector_DINT);
NodeFactory.AddNodeAsPrototype('Vision/Constants/ContainerType_Vector_UDINT', node_ContainerType_Vector_UDINT);
NodeFactory.AddNodeAsPrototype('Vision/Constants/ContainerType_Vector_ULINT', node_ContainerType_Vector_ULINT);
NodeFactory.AddNodeAsPrototype('Vision/Constants/ContainerType_Vector_REAL', node_ContainerType_Vector_REAL);
NodeFactory.AddNodeAsPrototype('Vision/Constants/ContainerType_Vector_LREAL', node_ContainerType_Vector_LREAL);
NodeFactory.AddNodeAsPrototype('Vision/Constants/ContainerType_Vector_ITcVnImage', node_ContainerType_Vector_ITcVnImage);
NodeFactory.AddNodeAsPrototype('Vision/Constants/ContainerType_Vector_TcVnPoint2_DINT', node_ContainerType_Vector_TcVnPoint2_DINT);
NodeFactory.AddNodeAsPrototype('Vision/Constants/ContainerType_Vector_TcVnPoint2_REAL', node_ContainerType_Vector_TcVnPoint2_REAL);
NodeFactory.AddNodeAsPrototype('Vision/Constants/ContainerType_Vector_TcVnPoint2_LREAL', node_ContainerType_Vector_TcVnPoint2_LREAL);
NodeFactory.AddNodeAsPrototype('Vision/Constants/ContainerType_Vector_TcVnPoint3_REAL', node_ContainerType_Vector_TcVnPoint3_REAL);
NodeFactory.AddNodeAsPrototype('Vision/Constants/ContainerType_Vector_TcVnPoint3_LREAL', node_ContainerType_Vector_TcVnPoint3_LREAL);
NodeFactory.AddNodeAsPrototype('Vision/Constants/ContainerType_Vector_Vector_TcVnPoint2_DINT', node_ContainerType_Vector_Vector_TcVnPoint2_DINT);
NodeFactory.AddNodeAsPrototype('Vision/Constants/ContainerType_Vector_Vector_TcVnPoint2_REAL', node_ContainerType_Vector_Vector_TcVnPoint2_REAL);
NodeFactory.AddNodeAsPrototype('Vision/Constants/ContainerType_Vector_Vector_TcVnPoint3_REAL', node_ContainerType_Vector_Vector_TcVnPoint3_REAL);
NodeFactory.AddNodeAsPrototype('Vision/Constants/ContainerType_Vector_Vector_UDINT', node_ContainerType_Vector_Vector_UDINT);
NodeFactory.AddNodeAsPrototype('Vision/Constants/ContainerType_Vector_Vector_ULINT', node_ContainerType_Vector_Vector_ULINT);
NodeFactory.AddNodeAsPrototype('Vision/Constants/ContainerType_Vector_Vector_REAL', node_ContainerType_Vector_Vector_REAL);
NodeFactory.AddNodeAsPrototype('Vision/Constants/ContainerType_Vector_Vector_LREAL', node_ContainerType_Vector_Vector_LREAL);
NodeFactory.AddNodeAsPrototype('Vision/Constants/ContainerType_Vector_TcVnVector2_SINT', node_ContainerType_Vector_TcVnVector2_SINT);
NodeFactory.AddNodeAsPrototype('Vision/Constants/ContainerType_Vector_TcVnVector2_USINT', node_ContainerType_Vector_TcVnVector2_USINT);
NodeFactory.AddNodeAsPrototype('Vision/Constants/ContainerType_Vector_TcVnVector2_INT', node_ContainerType_Vector_TcVnVector2_INT);
NodeFactory.AddNodeAsPrototype('Vision/Constants/ContainerType_Vector_TcVnVector2_UINT', node_ContainerType_Vector_TcVnVector2_UINT);
NodeFactory.AddNodeAsPrototype('Vision/Constants/ContainerType_Vector_TcVnVector2_DINT', node_ContainerType_Vector_TcVnVector2_DINT);
NodeFactory.AddNodeAsPrototype('Vision/Constants/ContainerType_Vector_TcVnVector2_REAL', node_ContainerType_Vector_TcVnVector2_REAL);
NodeFactory.AddNodeAsPrototype('Vision/Constants/ContainerType_Vector_TcVnVector3_SINT', node_ContainerType_Vector_TcVnVector3_SINT);
NodeFactory.AddNodeAsPrototype('Vision/Constants/ContainerType_Vector_TcVnVector3_USINT', node_ContainerType_Vector_TcVnVector3_USINT);
NodeFactory.AddNodeAsPrototype('Vision/Constants/ContainerType_Vector_TcVnVector3_INT', node_ContainerType_Vector_TcVnVector3_INT);
NodeFactory.AddNodeAsPrototype('Vision/Constants/ContainerType_Vector_TcVnVector3_UINT', node_ContainerType_Vector_TcVnVector3_UINT);
NodeFactory.AddNodeAsPrototype('Vision/Constants/ContainerType_Vector_TcVnVector3_REAL', node_ContainerType_Vector_TcVnVector3_REAL);
NodeFactory.AddNodeAsPrototype('Vision/Constants/ContainerType_Vector_TcVnVector4_SINT', node_ContainerType_Vector_TcVnVector4_SINT);
NodeFactory.AddNodeAsPrototype('Vision/Constants/ContainerType_Vector_TcVnVector4_USINT', node_ContainerType_Vector_TcVnVector4_USINT);
NodeFactory.AddNodeAsPrototype('Vision/Constants/ContainerType_Vector_TcVnVector4_INT', node_ContainerType_Vector_TcVnVector4_INT);
NodeFactory.AddNodeAsPrototype('Vision/Constants/ContainerType_Vector_TcVnVector4_UINT', node_ContainerType_Vector_TcVnVector4_UINT);
NodeFactory.AddNodeAsPrototype('Vision/Constants/ContainerType_Vector_TcVnVector4_DINT', node_ContainerType_Vector_TcVnVector4_DINT);
NodeFactory.AddNodeAsPrototype('Vision/Constants/ContainerType_Vector_TcVnVector4_REAL', node_ContainerType_Vector_TcVnVector4_REAL);
NodeFactory.AddNodeAsPrototype('Vision/Constants/ContainerType_Vector_TcVnVector4_LREAL', node_ContainerType_Vector_TcVnVector4_LREAL);
NodeFactory.AddNodeAsPrototype('Vision/Constants/ContainerType_Vector_TcVnRectangle_DINT', node_ContainerType_Vector_TcVnRectangle_DINT);
NodeFactory.AddNodeAsPrototype('Vision/Constants/ContainerType_Vector_TcVnRotatedRectangle', node_ContainerType_Vector_TcVnRotatedRectangle);
NodeFactory.AddNodeAsPrototype('Vision/Constants/ContainerType_Vector_TcVnKeyPoint', node_ContainerType_Vector_TcVnKeyPoint);
NodeFactory.AddNodeAsPrototype('Vision/Constants/ContainerType_Vector_TcVnDMatch', node_ContainerType_Vector_TcVnDMatch);
NodeFactory.AddNodeAsPrototype('Vision/Constants/ContainerType_Vector_Vector_TcVnDMatch', node_ContainerType_Vector_Vector_TcVnDMatch);
NodeFactory.AddNodeAsPrototype('Vision/Constants/ContainerType_String_SINT', node_ContainerType_String_SINT);
NodeFactory.AddNodeAsPrototype('Vision/Constants/ContainerType_Vector_String_SINT', node_ContainerType_Vector_String_SINT);

// Container Statistics
NodeFactory.AddNodeAsPrototype('Vision/Container Statistics/F_VN_MaxElementElementwise/F_VN_MaxElementElementwise_DINT', node_F_VN_MaxElementElementwise_DINT);
NodeFactory.AddNodeAsPrototype('Vision/Container Statistics/F_VN_MaxElementElementwise/F_VN_MaxElementElementwise_INT', node_F_VN_MaxElementElementwise_INT);
NodeFactory.AddNodeAsPrototype('Vision/Container Statistics/F_VN_MaxElementElementwise/F_VN_MaxElementElementwise_LREAL', node_F_VN_MaxElementElementwise_LREAL);
NodeFactory.AddNodeAsPrototype('Vision/Container Statistics/F_VN_MaxElementElementwise/F_VN_MaxElementElementwise_REAL', node_F_VN_MaxElementElementwise_REAL);
NodeFactory.AddNodeAsPrototype('Vision/Container Statistics/F_VN_MaxElementElementwise/F_VN_MaxElementElementwise_SINT', node_F_VN_MaxElementElementwise_SINT);
NodeFactory.AddNodeAsPrototype('Vision/Container Statistics/F_VN_MaxElementElementwise/F_VN_MaxElementElementwise_TcVnPoint2_DINT', node_F_VN_MaxElementElementwise_TcVnPoint2_DINT);
NodeFactory.AddNodeAsPrototype('Vision/Container Statistics/F_VN_MaxElementElementwise/F_VN_MaxElementElementwise_TcVnPoint2_LREAL', node_F_VN_MaxElementElementwise_TcVnPoint2_LREAL);
NodeFactory.AddNodeAsPrototype('Vision/Container Statistics/F_VN_MaxElementElementwise/F_VN_MaxElementElementwise_TcVnPoint2_REAL', node_F_VN_MaxElementElementwise_TcVnPoint2_REAL);
NodeFactory.AddNodeAsPrototype('Vision/Container Statistics/F_VN_MaxElementElementwise/F_VN_MaxElementElementwise_TcVnPoint3_LREAL', node_F_VN_MaxElementElementwise_TcVnPoint3_LREAL);
NodeFactory.AddNodeAsPrototype('Vision/Container Statistics/F_VN_MaxElementElementwise/F_VN_MaxElementElementwise_TcVnPoint3_REAL', node_F_VN_MaxElementElementwise_TcVnPoint3_REAL);
NodeFactory.AddNodeAsPrototype('Vision/Container Statistics/F_VN_MaxElementElementwise/F_VN_MaxElementElementwise_TcVnVector2_DINT', node_F_VN_MaxElementElementwise_TcVnVector2_DINT);
NodeFactory.AddNodeAsPrototype('Vision/Container Statistics/F_VN_MaxElementElementwise/F_VN_MaxElementElementwise_TcVnVector2_INT', node_F_VN_MaxElementElementwise_TcVnVector2_INT);
NodeFactory.AddNodeAsPrototype('Vision/Container Statistics/F_VN_MaxElementElementwise/F_VN_MaxElementElementwise_TcVnVector2_REAL', node_F_VN_MaxElementElementwise_TcVnVector2_REAL);
NodeFactory.AddNodeAsPrototype('Vision/Container Statistics/F_VN_MaxElementElementwise/F_VN_MaxElementElementwise_TcVnVector2_SINT', node_F_VN_MaxElementElementwise_TcVnVector2_SINT);
NodeFactory.AddNodeAsPrototype('Vision/Container Statistics/F_VN_MaxElementElementwise/F_VN_MaxElementElementwise_TcVnVector2_UINT', node_F_VN_MaxElementElementwise_TcVnVector2_UINT);
NodeFactory.AddNodeAsPrototype('Vision/Container Statistics/F_VN_MaxElementElementwise/F_VN_MaxElementElementwise_TcVnVector2_USINT', node_F_VN_MaxElementElementwise_TcVnVector2_USINT);
NodeFactory.AddNodeAsPrototype('Vision/Container Statistics/F_VN_MaxElementElementwise/F_VN_MaxElementElementwise_TcVnVector3_INT', node_F_VN_MaxElementElementwise_TcVnVector3_INT);
NodeFactory.AddNodeAsPrototype('Vision/Container Statistics/F_VN_MaxElementElementwise/F_VN_MaxElementElementwise_TcVnVector3_REAL', node_F_VN_MaxElementElementwise_TcVnVector3_REAL);
NodeFactory.AddNodeAsPrototype('Vision/Container Statistics/F_VN_MaxElementElementwise/F_VN_MaxElementElementwise_TcVnVector3_SINT', node_F_VN_MaxElementElementwise_TcVnVector3_SINT);
NodeFactory.AddNodeAsPrototype('Vision/Container Statistics/F_VN_MaxElementElementwise/F_VN_MaxElementElementwise_TcVnVector3_UINT', node_F_VN_MaxElementElementwise_TcVnVector3_UINT);
NodeFactory.AddNodeAsPrototype('Vision/Container Statistics/F_VN_MaxElementElementwise/F_VN_MaxElementElementwise_TcVnVector3_USINT', node_F_VN_MaxElementElementwise_TcVnVector3_USINT);
NodeFactory.AddNodeAsPrototype('Vision/Container Statistics/F_VN_MaxElementElementwise/F_VN_MaxElementElementwise_TcVnVector4_DINT', node_F_VN_MaxElementElementwise_TcVnVector4_DINT);
NodeFactory.AddNodeAsPrototype('Vision/Container Statistics/F_VN_MaxElementElementwise/F_VN_MaxElementElementwise_TcVnVector4_INT', node_F_VN_MaxElementElementwise_TcVnVector4_INT);
NodeFactory.AddNodeAsPrototype('Vision/Container Statistics/F_VN_MaxElementElementwise/F_VN_MaxElementElementwise_TcVnVector4_LREAL', node_F_VN_MaxElementElementwise_TcVnVector4_LREAL);
NodeFactory.AddNodeAsPrototype('Vision/Container Statistics/F_VN_MaxElementElementwise/F_VN_MaxElementElementwise_TcVnVector4_REAL', node_F_VN_MaxElementElementwise_TcVnVector4_REAL);
NodeFactory.AddNodeAsPrototype('Vision/Container Statistics/F_VN_MaxElementElementwise/F_VN_MaxElementElementwise_TcVnVector4_SINT', node_F_VN_MaxElementElementwise_TcVnVector4_SINT);
NodeFactory.AddNodeAsPrototype('Vision/Container Statistics/F_VN_MaxElementElementwise/F_VN_MaxElementElementwise_TcVnVector4_UINT', node_F_VN_MaxElementElementwise_TcVnVector4_UINT);
NodeFactory.AddNodeAsPrototype('Vision/Container Statistics/F_VN_MaxElementElementwise/F_VN_MaxElementElementwise_TcVnVector4_USINT', node_F_VN_MaxElementElementwise_TcVnVector4_USINT);
NodeFactory.AddNodeAsPrototype('Vision/Container Statistics/F_VN_MaxElementElementwise/F_VN_MaxElementElementwise_UDINT', node_F_VN_MaxElementElementwise_UDINT);
NodeFactory.AddNodeAsPrototype('Vision/Container Statistics/F_VN_MaxElementElementwise/F_VN_MaxElementElementwise_UINT', node_F_VN_MaxElementElementwise_UINT);
NodeFactory.AddNodeAsPrototype('Vision/Container Statistics/F_VN_MaxElementElementwise/F_VN_MaxElementElementwise_ULINT', node_F_VN_MaxElementElementwise_ULINT);
NodeFactory.AddNodeAsPrototype('Vision/Container Statistics/F_VN_MaxElementElementwise/F_VN_MaxElementElementwise_USINT', node_F_VN_MaxElementElementwise_USINT);

NodeFactory.AddNodeAsPrototype('Vision/Container Statistics/F_VN_MedianElementElementwise/F_VN_MedianElementElementwise_DINT', node_F_VN_MedianElementElementwise_DINT);
NodeFactory.AddNodeAsPrototype('Vision/Container Statistics/F_VN_MedianElementElementwise/F_VN_MedianElementElementwise_INT', node_F_VN_MedianElementElementwise_INT);
NodeFactory.AddNodeAsPrototype('Vision/Container Statistics/F_VN_MedianElementElementwise/F_VN_MedianElementElementwise_LREAL', node_F_VN_MedianElementElementwise_LREAL);
NodeFactory.AddNodeAsPrototype('Vision/Container Statistics/F_VN_MedianElementElementwise/F_VN_MedianElementElementwise_REAL', node_F_VN_MedianElementElementwise_REAL);
NodeFactory.AddNodeAsPrototype('Vision/Container Statistics/F_VN_MedianElementElementwise/F_VN_MedianElementElementwise_SINT', node_F_VN_MedianElementElementwise_SINT);
NodeFactory.AddNodeAsPrototype('Vision/Container Statistics/F_VN_MedianElementElementwise/F_VN_MedianElementElementwise_TcVnPoint2_DINT', node_F_VN_MedianElementElementwise_TcVnPoint2_DINT);
NodeFactory.AddNodeAsPrototype('Vision/Container Statistics/F_VN_MedianElementElementwise/F_VN_MedianElementElementwise_TcVnPoint2_LREAL', node_F_VN_MedianElementElementwise_TcVnPoint2_LREAL);
NodeFactory.AddNodeAsPrototype('Vision/Container Statistics/F_VN_MedianElementElementwise/F_VN_MedianElementElementwise_TcVnPoint2_REAL', node_F_VN_MedianElementElementwise_TcVnPoint2_REAL);
NodeFactory.AddNodeAsPrototype('Vision/Container Statistics/F_VN_MedianElementElementwise/F_VN_MedianElementElementwise_TcVnPoint3_LREAL', node_F_VN_MedianElementElementwise_TcVnPoint3_LREAL);
NodeFactory.AddNodeAsPrototype('Vision/Container Statistics/F_VN_MedianElementElementwise/F_VN_MedianElementElementwise_TcVnPoint3_REAL', node_F_VN_MedianElementElementwise_TcVnPoint3_REAL);
NodeFactory.AddNodeAsPrototype('Vision/Container Statistics/F_VN_MedianElementElementwise/F_VN_MedianElementElementwise_TcVnVector2_DINT', node_F_VN_MedianElementElementwise_TcVnVector2_DINT);
NodeFactory.AddNodeAsPrototype('Vision/Container Statistics/F_VN_MedianElementElementwise/F_VN_MedianElementElementwise_TcVnVector2_INT', node_F_VN_MedianElementElementwise_TcVnVector2_INT);
NodeFactory.AddNodeAsPrototype('Vision/Container Statistics/F_VN_MedianElementElementwise/F_VN_MedianElementElementwise_TcVnVector2_REAL', node_F_VN_MedianElementElementwise_TcVnVector2_REAL);
NodeFactory.AddNodeAsPrototype('Vision/Container Statistics/F_VN_MedianElementElementwise/F_VN_MedianElementElementwise_TcVnVector2_SINT', node_F_VN_MedianElementElementwise_TcVnVector2_SINT);
NodeFactory.AddNodeAsPrototype('Vision/Container Statistics/F_VN_MedianElementElementwise/F_VN_MedianElementElementwise_TcVnVector2_UINT', node_F_VN_MedianElementElementwise_TcVnVector2_UINT);
NodeFactory.AddNodeAsPrototype('Vision/Container Statistics/F_VN_MedianElementElementwise/F_VN_MedianElementElementwise_TcVnVector2_USINT', node_F_VN_MedianElementElementwise_TcVnVector2_USINT);
NodeFactory.AddNodeAsPrototype('Vision/Container Statistics/F_VN_MedianElementElementwise/F_VN_MedianElementElementwise_TcVnVector3_INT', node_F_VN_MedianElementElementwise_TcVnVector3_INT);
NodeFactory.AddNodeAsPrototype('Vision/Container Statistics/F_VN_MedianElementElementwise/F_VN_MedianElementElementwise_TcVnVector3_REAL', node_F_VN_MedianElementElementwise_TcVnVector3_REAL);
NodeFactory.AddNodeAsPrototype('Vision/Container Statistics/F_VN_MedianElementElementwise/F_VN_MedianElementElementwise_TcVnVector3_SINT', node_F_VN_MedianElementElementwise_TcVnVector3_SINT);
NodeFactory.AddNodeAsPrototype('Vision/Container Statistics/F_VN_MedianElementElementwise/F_VN_MedianElementElementwise_TcVnVector3_UINT', node_F_VN_MedianElementElementwise_TcVnVector3_UINT);
NodeFactory.AddNodeAsPrototype('Vision/Container Statistics/F_VN_MedianElementElementwise/F_VN_MedianElementElementwise_TcVnVector3_USINT', node_F_VN_MedianElementElementwise_TcVnVector3_USINT);
NodeFactory.AddNodeAsPrototype('Vision/Container Statistics/F_VN_MedianElementElementwise/F_VN_MedianElementElementwise_TcVnVector4_DINT', node_F_VN_MedianElementElementwise_TcVnVector4_DINT);
NodeFactory.AddNodeAsPrototype('Vision/Container Statistics/F_VN_MedianElementElementwise/F_VN_MedianElementElementwise_TcVnVector4_INT', node_F_VN_MedianElementElementwise_TcVnVector4_INT);
NodeFactory.AddNodeAsPrototype('Vision/Container Statistics/F_VN_MedianElementElementwise/F_VN_MedianElementElementwise_TcVnVector4_LREAL', node_F_VN_MedianElementElementwise_TcVnVector4_LREAL);
NodeFactory.AddNodeAsPrototype('Vision/Container Statistics/F_VN_MedianElementElementwise/F_VN_MedianElementElementwise_TcVnVector4_REAL', node_F_VN_MedianElementElementwise_TcVnVector4_REAL);
NodeFactory.AddNodeAsPrototype('Vision/Container Statistics/F_VN_MedianElementElementwise/F_VN_MedianElementElementwise_TcVnVector4_SINT', node_F_VN_MedianElementElementwise_TcVnVector4_SINT);
NodeFactory.AddNodeAsPrototype('Vision/Container Statistics/F_VN_MedianElementElementwise/F_VN_MedianElementElementwise_TcVnVector4_UINT', node_F_VN_MedianElementElementwise_TcVnVector4_UINT);
NodeFactory.AddNodeAsPrototype('Vision/Container Statistics/F_VN_MedianElementElementwise/F_VN_MedianElementElementwise_TcVnVector4_USINT', node_F_VN_MedianElementElementwise_TcVnVector4_USINT);
NodeFactory.AddNodeAsPrototype('Vision/Container Statistics/F_VN_MedianElementElementwise/F_VN_MedianElementElementwise_UDINT', node_F_VN_MedianElementElementwise_UDINT);
NodeFactory.AddNodeAsPrototype('Vision/Container Statistics/F_VN_MedianElementElementwise/F_VN_MedianElementElementwise_UINT', node_F_VN_MedianElementElementwise_UINT);
NodeFactory.AddNodeAsPrototype('Vision/Container Statistics/F_VN_MedianElementElementwise/F_VN_MedianElementElementwise_ULINT', node_F_VN_MedianElementElementwise_ULINT);
NodeFactory.AddNodeAsPrototype('Vision/Container Statistics/F_VN_MedianElementElementwise/F_VN_MedianElementElementwise_USINT', node_F_VN_MedianElementElementwise_USINT);

NodeFactory.AddNodeAsPrototype('Vision/Container Statistics/F_VN_MinElementElementwise/F_VN_MinElementElementwise_DINT', node_F_VN_MinElementElementwise_DINT);
NodeFactory.AddNodeAsPrototype('Vision/Container Statistics/F_VN_MinElementElementwise/F_VN_MinElementElementwise_INT', node_F_VN_MinElementElementwise_INT);
NodeFactory.AddNodeAsPrototype('Vision/Container Statistics/F_VN_MinElementElementwise/F_VN_MinElementElementwise_LREAL', node_F_VN_MinElementElementwise_LREAL);
NodeFactory.AddNodeAsPrototype('Vision/Container Statistics/F_VN_MinElementElementwise/F_VN_MinElementElementwise_REAL', node_F_VN_MinElementElementwise_REAL);
NodeFactory.AddNodeAsPrototype('Vision/Container Statistics/F_VN_MinElementElementwise/F_VN_MinElementElementwise_SINT', node_F_VN_MinElementElementwise_SINT);
NodeFactory.AddNodeAsPrototype('Vision/Container Statistics/F_VN_MinElementElementwise/F_VN_MinElementElementwise_TcVnPoint2_DINT', node_F_VN_MinElementElementwise_TcVnPoint2_DINT);
NodeFactory.AddNodeAsPrototype('Vision/Container Statistics/F_VN_MinElementElementwise/F_VN_MinElementElementwise_TcVnPoint2_LREAL', node_F_VN_MinElementElementwise_TcVnPoint2_LREAL);
NodeFactory.AddNodeAsPrototype('Vision/Container Statistics/F_VN_MinElementElementwise/F_VN_MinElementElementwise_TcVnPoint2_REAL', node_F_VN_MinElementElementwise_TcVnPoint2_REAL);
NodeFactory.AddNodeAsPrototype('Vision/Container Statistics/F_VN_MinElementElementwise/F_VN_MinElementElementwise_TcVnPoint3_LREAL', node_F_VN_MinElementElementwise_TcVnPoint3_LREAL);
NodeFactory.AddNodeAsPrototype('Vision/Container Statistics/F_VN_MinElementElementwise/F_VN_MinElementElementwise_TcVnPoint3_REAL', node_F_VN_MinElementElementwise_TcVnPoint3_REAL);
NodeFactory.AddNodeAsPrototype('Vision/Container Statistics/F_VN_MinElementElementwise/F_VN_MinElementElementwise_TcVnVector2_DINT', node_F_VN_MinElementElementwise_TcVnVector2_DINT);
NodeFactory.AddNodeAsPrototype('Vision/Container Statistics/F_VN_MinElementElementwise/F_VN_MinElementElementwise_TcVnVector2_INT', node_F_VN_MinElementElementwise_TcVnVector2_INT);
NodeFactory.AddNodeAsPrototype('Vision/Container Statistics/F_VN_MinElementElementwise/F_VN_MinElementElementwise_TcVnVector2_REAL', node_F_VN_MinElementElementwise_TcVnVector2_REAL);
NodeFactory.AddNodeAsPrototype('Vision/Container Statistics/F_VN_MinElementElementwise/F_VN_MinElementElementwise_TcVnVector2_SINT', node_F_VN_MinElementElementwise_TcVnVector2_SINT);
NodeFactory.AddNodeAsPrototype('Vision/Container Statistics/F_VN_MinElementElementwise/F_VN_MinElementElementwise_TcVnVector2_UINT', node_F_VN_MinElementElementwise_TcVnVector2_UINT);
NodeFactory.AddNodeAsPrototype('Vision/Container Statistics/F_VN_MinElementElementwise/F_VN_MinElementElementwise_TcVnVector2_USINT', node_F_VN_MinElementElementwise_TcVnVector2_USINT);
NodeFactory.AddNodeAsPrototype('Vision/Container Statistics/F_VN_MinElementElementwise/F_VN_MinElementElementwise_TcVnVector3_INT', node_F_VN_MinElementElementwise_TcVnVector3_INT);
NodeFactory.AddNodeAsPrototype('Vision/Container Statistics/F_VN_MinElementElementwise/F_VN_MinElementElementwise_TcVnVector3_REAL', node_F_VN_MinElementElementwise_TcVnVector3_REAL);
NodeFactory.AddNodeAsPrototype('Vision/Container Statistics/F_VN_MinElementElementwise/F_VN_MinElementElementwise_TcVnVector3_SINT', node_F_VN_MinElementElementwise_TcVnVector3_SINT);
NodeFactory.AddNodeAsPrototype('Vision/Container Statistics/F_VN_MinElementElementwise/F_VN_MinElementElementwise_TcVnVector3_UINT', node_F_VN_MinElementElementwise_TcVnVector3_UINT);
NodeFactory.AddNodeAsPrototype('Vision/Container Statistics/F_VN_MinElementElementwise/F_VN_MinElementElementwise_TcVnVector3_USINT', node_F_VN_MinElementElementwise_TcVnVector3_USINT);
NodeFactory.AddNodeAsPrototype('Vision/Container Statistics/F_VN_MinElementElementwise/F_VN_MinElementElementwise_TcVnVector4_DINT', node_F_VN_MinElementElementwise_TcVnVector4_DINT);
NodeFactory.AddNodeAsPrototype('Vision/Container Statistics/F_VN_MinElementElementwise/F_VN_MinElementElementwise_TcVnVector4_INT', node_F_VN_MinElementElementwise_TcVnVector4_INT);
NodeFactory.AddNodeAsPrototype('Vision/Container Statistics/F_VN_MinElementElementwise/F_VN_MinElementElementwise_TcVnVector4_LREAL', node_F_VN_MinElementElementwise_TcVnVector4_LREAL);
NodeFactory.AddNodeAsPrototype('Vision/Container Statistics/F_VN_MinElementElementwise/F_VN_MinElementElementwise_TcVnVector4_REAL', node_F_VN_MinElementElementwise_TcVnVector4_REAL);
NodeFactory.AddNodeAsPrototype('Vision/Container Statistics/F_VN_MinElementElementwise/F_VN_MinElementElementwise_TcVnVector4_SINT', node_F_VN_MinElementElementwise_TcVnVector4_SINT);
NodeFactory.AddNodeAsPrototype('Vision/Container Statistics/F_VN_MinElementElementwise/F_VN_MinElementElementwise_TcVnVector4_UINT', node_F_VN_MinElementElementwise_TcVnVector4_UINT);
NodeFactory.AddNodeAsPrototype('Vision/Container Statistics/F_VN_MinElementElementwise/F_VN_MinElementElementwise_TcVnVector4_USINT', node_F_VN_MinElementElementwise_TcVnVector4_USINT);
NodeFactory.AddNodeAsPrototype('Vision/Container Statistics/F_VN_MinElementElementwise/F_VN_MinElementElementwise_UDINT', node_F_VN_MinElementElementwise_UDINT);
NodeFactory.AddNodeAsPrototype('Vision/Container Statistics/F_VN_MinElementElementwise/F_VN_MinElementElementwise_UINT', node_F_VN_MinElementElementwise_UINT);
NodeFactory.AddNodeAsPrototype('Vision/Container Statistics/F_VN_MinElementElementwise/F_VN_MinElementElementwise_ULINT', node_F_VN_MinElementElementwise_ULINT);
NodeFactory.AddNodeAsPrototype('Vision/Container Statistics/F_VN_MinElementElementwise/F_VN_MinElementElementwise_USINT', node_F_VN_MinElementElementwise_USINT);
NodeFactory.AddNodeAsPrototype('Vision/Container Statistics/F_VN_ContainerAverage', node_F_VN_ContainerAverage);
NodeFactory.AddNodeAsPrototype('Vision/Container Statistics/F_VN_ContainerAverageElementwise2', node_F_VN_ContainerAverageElementwise2);
NodeFactory.AddNodeAsPrototype('Vision/Container Statistics/F_VN_ContainerAverageElementwise3', node_F_VN_ContainerAverageElementwise3);
NodeFactory.AddNodeAsPrototype('Vision/Container Statistics/F_VN_ContainerAverageElementwise4', node_F_VN_ContainerAverageElementwise4);
NodeFactory.AddNodeAsPrototype('Vision/Container Statistics/F_VN_ContainerAverageVariance', node_F_VN_ContainerAverageVariance);
NodeFactory.AddNodeAsPrototype('Vision/Container Statistics/F_VN_ContainerAverageVarianceElementwise2', node_F_VN_ContainerAverageVarianceElementwise2);
NodeFactory.AddNodeAsPrototype('Vision/Container Statistics/F_VN_ContainerAverageVarianceElementwise3', node_F_VN_ContainerAverageVarianceElementwise3);
NodeFactory.AddNodeAsPrototype('Vision/Container Statistics/F_VN_ContainerAverageVarianceElementwise4', node_F_VN_ContainerAverageVarianceElementwise4);
NodeFactory.AddNodeAsPrototype('Vision/Container Statistics/F_VN_MaxElement', node_F_VN_MaxElement);
NodeFactory.AddNodeAsPrototype('Vision/Container Statistics/F_VN_MedianElement', node_F_VN_MedianElement);
NodeFactory.AddNodeAsPrototype('Vision/Container Statistics/F_VN_MinElement', node_F_VN_MinElement);

// Contour Analysis
NodeFactory.AddNodeAsPrototype('Vision/Contour Analysis/F_VN_ApproximatePolygon', node_F_VN_ApproximatePolygon);
NodeFactory.AddNodeAsPrototype('Vision/Contour Analysis/F_VN_CheckIfPointIsInsideContour', node_F_VN_CheckIfPointIsInsideContour);
NodeFactory.AddNodeAsPrototype('Vision/Contour Analysis/F_VN_ContourArea', node_F_VN_ContourArea);
NodeFactory.AddNodeAsPrototype('Vision/Contour Analysis/F_VN_ContourCenterOfMass', node_F_VN_ContourCenterOfMass);
NodeFactory.AddNodeAsPrototype('Vision/Contour Analysis/F_VN_ContourCircularity', node_F_VN_ContourCircularity);
NodeFactory.AddNodeAsPrototype('Vision/Contour Analysis/F_VN_ContourCircularityExp', node_F_VN_ContourCircularityExp);
NodeFactory.AddNodeAsPrototype('Vision/Contour Analysis/F_VN_ContourConvexity', node_F_VN_ContourConvexity);
NodeFactory.AddNodeAsPrototype('Vision/Contour Analysis/F_VN_ContourEccentricity', node_F_VN_ContourEccentricity);
NodeFactory.AddNodeAsPrototype('Vision/Contour Analysis/F_VN_ContourElongation', node_F_VN_ContourElongation);
NodeFactory.AddNodeAsPrototype('Vision/Contour Analysis/F_VN_ContourExtremePoint', node_F_VN_ContourExtremePoint);
NodeFactory.AddNodeAsPrototype('Vision/Contour Analysis/F_VN_ContourInertiaRatio', node_F_VN_ContourInertiaRatio);
NodeFactory.AddNodeAsPrototype('Vision/Contour Analysis/F_VN_ContourMoments', node_F_VN_ContourMoments);
NodeFactory.AddNodeAsPrototype('Vision/Contour Analysis/F_VN_ContourOrientation', node_F_VN_ContourOrientation);
NodeFactory.AddNodeAsPrototype('Vision/Contour Analysis/F_VN_ContourOrientationExp', node_F_VN_ContourOrientationExp);
NodeFactory.AddNodeAsPrototype('Vision/Contour Analysis/F_VN_ContourPerimeter', node_F_VN_ContourPerimeter);
NodeFactory.AddNodeAsPrototype('Vision/Contour Analysis/F_VN_ContourRoundness', node_F_VN_ContourRoundness);
NodeFactory.AddNodeAsPrototype('Vision/Contour Analysis/F_VN_ConvexHullPoints', node_F_VN_ConvexHullPoints);
NodeFactory.AddNodeAsPrototype('Vision/Contour Analysis/F_VN_ConvexHullPointsExp', node_F_VN_ConvexHullPointsExp);
NodeFactory.AddNodeAsPrototype('Vision/Contour Analysis/F_VN_ConvexityDefects', node_F_VN_ConvexityDefects);
//NodeFactory.AddNodeAsPrototype('Vision/Contour Analysis/F_VN_CustomElementWiseContainerOperation_ITcVnContainer', node_F_VN_CustomElementWiseContainerOperation_ITcVnContainer);
//NodeFactory.AddNodeAsPrototype('Vision/Contour Analysis/F_VN_CustomElementWiseContainerOperation_ITcVnForwardIterator', node_F_VN_CustomElementWiseContainerOperation_ITcVnForwardIterator);
NodeFactory.AddNodeAsPrototype('Vision/Contour Analysis/F_VN_EnclosingCircle', node_F_VN_EnclosingCircle);
NodeFactory.AddNodeAsPrototype('Vision/Contour Analysis/F_VN_EnclosingRectangle', node_F_VN_EnclosingRectangle);
NodeFactory.AddNodeAsPrototype('Vision/Contour Analysis/F_VN_EnclosingTriangle', node_F_VN_EnclosingTriangle);
NodeFactory.AddNodeAsPrototype('Vision/Contour Analysis/F_VN_FitEllipse', node_F_VN_FitEllipse);
NodeFactory.AddNodeAsPrototype('Vision/Contour Analysis/F_VN_FitLine', node_F_VN_FitLine);
NodeFactory.AddNodeAsPrototype('Vision/Contour Analysis/F_VN_FitLineExp', node_F_VN_FitLineExp);
//NodeFactory.AddNodeAsPrototype('Vision/Contour Analysis/F_VN_FourierDescriptors', node_F_VN_FourierDescriptors);
NodeFactory.AddNodeAsPrototype('Vision/Contour Analysis/F_VN_MatchContours', node_F_VN_MatchContours);
NodeFactory.AddNodeAsPrototype('Vision/Contour Analysis/F_VN_MatchContours1vsN', node_F_VN_MatchContours1vsN);
NodeFactory.AddNodeAsPrototype('Vision/Contour Analysis/F_VN_MatchContours1vsNExp', node_F_VN_MatchContours1vsNExp);
NodeFactory.AddNodeAsPrototype('Vision/Contour Analysis/F_VN_MatchContoursExp', node_F_VN_MatchContoursExp);
NodeFactory.AddNodeAsPrototype('Vision/Contour Analysis/F_VN_UprightBoundingRectangle', node_F_VN_UprightBoundingRectangle);

// Control Functions
//NodeFactory.AddNodeAsPrototype('Vision/Control Functions/F_VN_StartAbsWatchdog', node_F_VN_StartAbsWatchdog);
//NodeFactory.AddNodeAsPrototype('Vision/Control Functions/F_VN_StartAbsWatchdogExp', node_F_VN_StartAbsWatchdogExp);
//NodeFactory.AddNodeAsPrototype('Vision/Control Functions/F_VN_StartRelWatchdog', node_F_VN_StartRelWatchdog);
//NodeFactory.AddNodeAsPrototype('Vision/Control Functions/F_VN_StartRelWatchdogExp', node_F_VN_StartRelWatchdogExp);
//NodeFactory.AddNodeAsPrototype('Vision/Control Functions/F_VN_StopWatchdog', node_F_VN_StopWatchdog);
    
// Drawing
NodeFactory.AddNodeAsPrototype('Vision/Drawing/F_VN_DrawArrow', node_F_VN_DrawArrow);
NodeFactory.AddNodeAsPrototype('Vision/Drawing/F_VN_DrawArrow_TcVnVector4_DINT', node_F_VN_DrawArrow_TcVnVector4_DINT);
NodeFactory.AddNodeAsPrototype('Vision/Drawing/F_VN_DrawArrowExp', node_F_VN_DrawArrowExp);
NodeFactory.AddNodeAsPrototype('Vision/Drawing/F_VN_DrawArrowExp_TcVnVector4_DINT', node_F_VN_DrawArrowExp_TcVnVector4_DINT);
NodeFactory.AddNodeAsPrototype('Vision/Drawing/F_VN_DrawCircle', node_F_VN_DrawCircle);
NodeFactory.AddNodeAsPrototype('Vision/Drawing/F_VN_DrawCircleExp', node_F_VN_DrawCircleExp);
NodeFactory.AddNodeAsPrototype('Vision/Drawing/F_VN_DrawCircles', node_F_VN_DrawCircles);
NodeFactory.AddNodeAsPrototype('Vision/Drawing/F_VN_DrawCirclesExp', node_F_VN_DrawCirclesExp);
NodeFactory.AddNodeAsPrototype('Vision/Drawing/F_VN_DrawCircularArc', node_F_VN_DrawCircularArc);
NodeFactory.AddNodeAsPrototype('Vision/Drawing/F_VN_DrawCircularArcExp', node_F_VN_DrawCircularArcExp);
NodeFactory.AddNodeAsPrototype('Vision/Drawing/F_VN_DrawComponents', node_F_VN_DrawComponents);
NodeFactory.AddNodeAsPrototype('Vision/Drawing/F_VN_DrawComponentsExp', node_F_VN_DrawComponentsExp);
NodeFactory.AddNodeAsPrototype('Vision/Drawing/F_VN_DrawContours', node_F_VN_DrawContours);
NodeFactory.AddNodeAsPrototype('Vision/Drawing/F_VN_DrawContoursExp', node_F_VN_DrawContoursExp);
NodeFactory.AddNodeAsPrototype('Vision/Drawing/F_VN_DrawEllipse', node_F_VN_DrawEllipse);
NodeFactory.AddNodeAsPrototype('Vision/Drawing/F_VN_DrawEllipseExp', node_F_VN_DrawEllipseExp);
NodeFactory.AddNodeAsPrototype('Vision/Drawing/F_VN_DrawKeypoints', node_F_VN_DrawKeypoints);
NodeFactory.AddNodeAsPrototype('Vision/Drawing/F_VN_DrawKeypointsExp', node_F_VN_DrawKeypointsExp);
NodeFactory.AddNodeAsPrototype('Vision/Drawing/F_VN_DrawLine', node_F_VN_DrawLine);
NodeFactory.AddNodeAsPrototype('Vision/Drawing/F_VN_DrawLine_TcVnVector4_DINT', node_F_VN_DrawLine_TcVnVector4_DINT);
NodeFactory.AddNodeAsPrototype('Vision/Drawing/F_VN_DrawLine_TcVnVector4_LREAL', node_F_VN_DrawLine_TcVnVector4_LREAL);
NodeFactory.AddNodeAsPrototype('Vision/Drawing/F_VN_DrawLineExp', node_F_VN_DrawLineExp);
NodeFactory.AddNodeAsPrototype('Vision/Drawing/F_VN_DrawLineExp_TcVnVector4_DINT', node_F_VN_DrawLineExp_TcVnVector4_DINT);
NodeFactory.AddNodeAsPrototype('Vision/Drawing/F_VN_DrawLineExp_TcVnVector4_LREAL', node_F_VN_DrawLineExp_TcVnVector4_LREAL);
NodeFactory.AddNodeAsPrototype('Vision/Drawing/F_VN_DrawLines', node_F_VN_DrawLines);
NodeFactory.AddNodeAsPrototype('Vision/Drawing/F_VN_DrawLinesExp', node_F_VN_DrawLinesExp);
NodeFactory.AddNodeAsPrototype('Vision/Drawing/F_VN_DrawMatches', node_F_VN_DrawMatches);
NodeFactory.AddNodeAsPrototype('Vision/Drawing/F_VN_DrawMatchesExp', node_F_VN_DrawMatchesExp);
NodeFactory.AddNodeAsPrototype('Vision/Drawing/F_VN_DrawOrientation', node_F_VN_DrawOrientation);
NodeFactory.AddNodeAsPrototype('Vision/Drawing/F_VN_DrawOrientationExp', node_F_VN_DrawOrientationExp);
NodeFactory.AddNodeAsPrototype('Vision/Drawing/F_VN_DrawPoint', node_F_VN_DrawPoint);
NodeFactory.AddNodeAsPrototype('Vision/Drawing/F_VN_DrawPointExp', node_F_VN_DrawPointExp);
NodeFactory.AddNodeAsPrototype('Vision/Drawing/F_VN_DrawPoints', node_F_VN_DrawPoints);
NodeFactory.AddNodeAsPrototype('Vision/Drawing/F_VN_DrawPointsExp', node_F_VN_DrawPointsExp);
NodeFactory.AddNodeAsPrototype('Vision/Drawing/F_VN_DrawPolygon', node_F_VN_DrawPolygon);
NodeFactory.AddNodeAsPrototype('Vision/Drawing/F_VN_DrawPolygonExp', node_F_VN_DrawPolygonExp);
NodeFactory.AddNodeAsPrototype('Vision/Drawing/F_VN_DrawRectangle', node_F_VN_DrawRectangle);
NodeFactory.AddNodeAsPrototype('Vision/Drawing/F_VN_DrawRectangle_TcVnRectangle_DINT', node_F_VN_DrawRectangle_TcVnRectangle_DINT);
NodeFactory.AddNodeAsPrototype('Vision/Drawing/F_VN_DrawRectangle_TcVnRectangle_UDINT', node_F_VN_DrawRectangle_TcVnRectangle_UDINT);
NodeFactory.AddNodeAsPrototype('Vision/Drawing/F_VN_DrawRotatedRectangle', node_F_VN_DrawRotatedRectangle);
NodeFactory.AddNodeAsPrototype('Vision/Drawing/F_VN_DrawRotatedRectangleExp', node_F_VN_DrawRotatedRectangleExp);
NodeFactory.AddNodeAsPrototype('Vision/Drawing/F_VN_FillCircle', node_F_VN_FillCircle);
NodeFactory.AddNodeAsPrototype('Vision/Drawing/F_VN_FillContours', node_F_VN_FillContours);
NodeFactory.AddNodeAsPrototype('Vision/Drawing/F_VN_FillEllipse', node_F_VN_FillEllipse);
NodeFactory.AddNodeAsPrototype('Vision/Drawing/F_VN_FillPolygon', node_F_VN_FillPolygon);
NodeFactory.AddNodeAsPrototype('Vision/Drawing/F_VN_FillRectangle', node_F_VN_FillRectangle);
NodeFactory.AddNodeAsPrototype('Vision/Drawing/F_VN_FillRotatedRectangle', node_F_VN_FillRotatedRectangle);
NodeFactory.AddNodeAsPrototype('Vision/Drawing/F_VN_PlotIntensityProfile', node_F_VN_PlotIntensityProfile);
NodeFactory.AddNodeAsPrototype('Vision/Drawing/F_VN_PlotIntensityProfileExp', node_F_VN_PlotIntensityProfileExp);
NodeFactory.AddNodeAsPrototype('Vision/Drawing/F_VN_PutLabel', node_F_VN_PutLabel);
NodeFactory.AddNodeAsPrototype('Vision/Drawing/F_VN_PutLabelExp', node_F_VN_PutLabelExp);
NodeFactory.AddNodeAsPrototype('Vision/Drawing/F_VN_PutText', node_F_VN_PutText);
NodeFactory.AddNodeAsPrototype('Vision/Drawing/F_VN_PutTextExp', node_F_VN_PutTextExp);

// Fourier Analysis
NodeFactory.AddNodeAsPrototype('Vision/Fourier Analysis/F_VN_CreateBandpassButterworthFilter', node_F_VN_CreateBandpassButterworthFilter);
NodeFactory.AddNodeAsPrototype('Vision/Fourier Analysis/F_VN_CreateBandpassGaussianFilter', node_F_VN_CreateBandpassGaussianFilter);
NodeFactory.AddNodeAsPrototype('Vision/Fourier Analysis/F_VN_CreateBandrejectButterworthFilter', node_F_VN_CreateBandrejectButterworthFilter);
NodeFactory.AddNodeAsPrototype('Vision/Fourier Analysis/F_VN_CreateBandrejectGaussianFilter', node_F_VN_CreateBandrejectGaussianFilter);
NodeFactory.AddNodeAsPrototype('Vision/Fourier Analysis/F_VN_CreateHighpassButterworthFilter', node_F_VN_CreateHighpassButterworthFilter);
NodeFactory.AddNodeAsPrototype('Vision/Fourier Analysis/F_VN_CreateHighpassGaussianFilter', node_F_VN_CreateHighpassGaussianFilter);
NodeFactory.AddNodeAsPrototype('Vision/Fourier Analysis/F_VN_CreateLowpassButterworthFilter', node_F_VN_CreateLowpassButterworthFilter);
NodeFactory.AddNodeAsPrototype('Vision/Fourier Analysis/F_VN_CreateLowpassGaussianFilter', node_F_VN_CreateLowpassGaussianFilter);
NodeFactory.AddNodeAsPrototype('Vision/Fourier Analysis/F_VN_Dft', node_F_VN_Dft);
NodeFactory.AddNodeAsPrototype('Vision/Fourier Analysis/F_VN_InverseDft', node_F_VN_InverseDft);
NodeFactory.AddNodeAsPrototype('Vision/Fourier Analysis/F_VN_OptimalDftSize', node_F_VN_OptimalDftSize);

// Geometric and Coordinate Transformations
NodeFactory.AddNodeAsPrototype('Vision/Geometric and Coordinate Transformations/Calibration/F_VN_CalibrateCamera', node_F_VN_CalibrateCamera);
//NodeFactory.AddNodeAsPrototype('Vision/Geometric and Coordinate Transformations/Calibration/F_VN_CalibrateCameraExp', node_F_VN_CalibrateCameraExp);
//NodeFactory.AddNodeAsPrototype('Vision/Geometric and Coordinate Transformations/Calibration/F_VN_CalibrateCameraExp2', node_F_VN_CalibrateCameraExp2);
//NodeFactory.AddNodeAsPrototype('Vision/Geometric and Coordinate Transformations/Calibration/F_VN_CalibrateCameraExp3', node_F_VN_CalibrateCameraExp3);
NodeFactory.AddNodeAsPrototype('Vision/Geometric and Coordinate Transformations/Calibration/F_VN_CalibrateCameraManually', node_F_VN_CalibrateCameraManually);
NodeFactory.AddNodeAsPrototype('Vision/Geometric and Coordinate Transformations/Calibration/F_VN_CalibrateCameraManuallyExp', node_F_VN_CalibrateCameraManuallyExp);
NodeFactory.AddNodeAsPrototype('Vision/Geometric and Coordinate Transformations/Calibration/F_VN_CalibrateCameraPlanar', node_F_VN_CalibrateCameraPlanar);
NodeFactory.AddNodeAsPrototype('Vision/Geometric and Coordinate Transformations/Calibration/F_VN_CalibrateCameraPlanarExp', node_F_VN_CalibrateCameraPlanarExp);
//NodeFactory.AddNodeAsPrototype('Vision/Geometric and Coordinate Transformations/Calibration/F_VN_CalibrateLinescanCamera', node_F_VN_CalibrateLinescanCamera);
//NodeFactory.AddNodeAsPrototype('Vision/Geometric and Coordinate Transformations/Calibration/F_VN_CalibrateLinescanCameraExp', node_F_VN_CalibrateLinescanCameraExp);
NodeFactory.AddNodeAsPrototype('Vision/Geometric and Coordinate Transformations/Calibration/F_VN_CompensateLensDistortion', node_F_VN_CompensateLensDistortion);
NodeFactory.AddNodeAsPrototype('Vision/Geometric and Coordinate Transformations/Calibration/F_VN_CompensateLensDistortionExp1', node_F_VN_CompensateLensDistortionExp1);
NodeFactory.AddNodeAsPrototype('Vision/Geometric and Coordinate Transformations/Calibration/F_VN_CompensateLensDistortionExp2', node_F_VN_CompensateLensDistortionExp2);
NodeFactory.AddNodeAsPrototype('Vision/Geometric and Coordinate Transformations/Calibration/F_VN_CompensateLensDistortionForPoints', node_F_VN_CompensateLensDistortionForPoints);
NodeFactory.AddNodeAsPrototype('Vision/Geometric and Coordinate Transformations/Calibration/F_VN_CompensateLensDistortionForPointsExp1', node_F_VN_CompensateLensDistortionForPointsExp1);
NodeFactory.AddNodeAsPrototype('Vision/Geometric and Coordinate Transformations/Calibration/F_VN_CompensateLensDistortionForPointsExp2', node_F_VN_CompensateLensDistortionForPointsExp2);
NodeFactory.AddNodeAsPrototype('Vision/Geometric and Coordinate Transformations/Calibration/F_VN_DetectPatternPoints', node_F_VN_DetectPatternPoints);
NodeFactory.AddNodeAsPrototype('Vision/Geometric and Coordinate Transformations/Calibration/F_VN_DetectPatternPointsExp', node_F_VN_DetectPatternPointsExp);
NodeFactory.AddNodeAsPrototype('Vision/Geometric and Coordinate Transformations/Calibration/F_VN_DetectPatternPoints2', node_F_VN_DetectPatternPoints2);
NodeFactory.AddNodeAsPrototype('Vision/Geometric and Coordinate Transformations/Calibration/F_VN_GenerateCalibrationPatternReferencePoints', node_F_VN_GenerateCalibrationPatternReferencePoints);
NodeFactory.AddNodeAsPrototype('Vision/Geometric and Coordinate Transformations/Calibration/F_VN_ImagePointsWorldDistance', node_F_VN_ImagePointsWorldDistance);
NodeFactory.AddNodeAsPrototype('Vision/Geometric and Coordinate Transformations/Calibration/F_VN_SolvePnP', node_F_VN_SolvePnP);
NodeFactory.AddNodeAsPrototype('Vision/Geometric and Coordinate Transformations/Calibration/F_VN_SolvePnPExp', node_F_VN_SolvePnPExp);
NodeFactory.AddNodeAsPrototype('Vision/Geometric and Coordinate Transformations/Calibration/F_VN_SortAxisAlignedPatternPoints', node_F_VN_SortAxisAlignedPatternPoints);
NodeFactory.AddNodeAsPrototype('Vision/Geometric and Coordinate Transformations/Calibration/F_VN_SortDetectedPatternPoints', node_F_VN_SortDetectedPatternPoints);
NodeFactory.AddNodeAsPrototype('Vision/Geometric and Coordinate Transformations/Calibration/F_VN_TransformCoordinatesImageToWorld_Container', node_F_VN_TransformCoordinatesImageToWorld_Container);
NodeFactory.AddNodeAsPrototype('Vision/Geometric and Coordinate Transformations/Calibration/F_VN_TransformCoordinatesImageToWorld_Point', node_F_VN_TransformCoordinatesImageToWorld_Point);
NodeFactory.AddNodeAsPrototype('Vision/Geometric and Coordinate Transformations/Calibration/F_VN_TransformCoordinatesPlanar_Container', node_F_VN_TransformCoordinatesPlanar_Container);
NodeFactory.AddNodeAsPrototype('Vision/Geometric and Coordinate Transformations/Calibration/F_VN_TransformCoordinatesPlanar_Point', node_F_VN_TransformCoordinatesPlanar_Point);
NodeFactory.AddNodeAsPrototype('Vision/Geometric and Coordinate Transformations/Calibration/F_VN_TransformCoordinatesWorldToImage_Container', node_F_VN_TransformCoordinatesWorldToImage_Container);
NodeFactory.AddNodeAsPrototype('Vision/Geometric and Coordinate Transformations/Calibration/F_VN_TransformCoordinatesWorldToImage_Point', node_F_VN_TransformCoordinatesWorldToImage_Point);
NodeFactory.AddNodeAsPrototype('Vision/Geometric and Coordinate Transformations/F_VN_AlignRotatedImageRegion', node_F_VN_AlignRotatedImageRegion);
NodeFactory.AddNodeAsPrototype('Vision/Geometric and Coordinate Transformations/F_VN_AlignRotatedImageRegionExp', node_F_VN_AlignRotatedImageRegionExp);
NodeFactory.AddNodeAsPrototype('Vision/Geometric and Coordinate Transformations/F_VN_ApplyRotationToAffineTransformation', node_F_VN_ApplyRotationToAffineTransformation);
NodeFactory.AddNodeAsPrototype('Vision/Geometric and Coordinate Transformations/F_VN_ApplyRotationToAffineTransformationExp', node_F_VN_ApplyRotationToAffineTransformationExp);
NodeFactory.AddNodeAsPrototype('Vision/Geometric and Coordinate Transformations/F_VN_ApplyScalingToAffineTransformation', node_F_VN_ApplyScalingToAffineTransformation);
NodeFactory.AddNodeAsPrototype('Vision/Geometric and Coordinate Transformations/F_VN_ApplyScalingToAffineTransformationExp', node_F_VN_ApplyScalingToAffineTransformationExp);
NodeFactory.AddNodeAsPrototype('Vision/Geometric and Coordinate Transformations/F_VN_ApplyTranslationToAffineTransformation', node_F_VN_ApplyTranslationToAffineTransformation);
NodeFactory.AddNodeAsPrototype('Vision/Geometric and Coordinate Transformations/F_VN_ApplyTranslationToAffineTransformationExp', node_F_VN_ApplyTranslationToAffineTransformationExp);
NodeFactory.AddNodeAsPrototype('Vision/Geometric and Coordinate Transformations/F_VN_ApplyYAxisInversionToAffineTransformation', node_F_VN_ApplyYAxisInversionToAffineTransformation);
NodeFactory.AddNodeAsPrototype('Vision/Geometric and Coordinate Transformations/F_VN_ApplyYAxisInversionToAffineTransformationExp', node_F_VN_ApplyYAxisInversionToAffineTransformationExp);
NodeFactory.AddNodeAsPrototype('Vision/Polarization/F_VN_DemosaicPolarizedImage', node_F_VN_DemosaicPolarizedImage);
NodeFactory.AddNodeAsPrototype('Vision/Polarization/F_VN_AngleAndDegreeOfLinearPolarization', node_F_VN_AngleAndDegreeOfLinearPolarization);
NodeFactory.AddNodeAsPrototype('Vision/Polarization/F_VN_PolarizedImageGlareReduction', node_F_VN_PolarizedImageGlareReduction);
NodeFactory.AddNodeAsPrototype('Vision/Geometric and Coordinate Transformations/F_VN_ConvertCartesianToPolarAngleImage', node_F_VN_ConvertCartesianToPolarAngleImage);
NodeFactory.AddNodeAsPrototype('Vision/Geometric and Coordinate Transformations/F_VN_ConvertCartesianToPolarAngleImageExp', node_F_VN_ConvertCartesianToPolarAngleImageExp);
NodeFactory.AddNodeAsPrototype('Vision/Geometric and Coordinate Transformations/F_VN_ConvertCartesianToPolarAngles', node_F_VN_ConvertCartesianToPolarAngles);
NodeFactory.AddNodeAsPrototype('Vision/Geometric and Coordinate Transformations/F_VN_ConvertCartesianToPolarAnglesExp', node_F_VN_ConvertCartesianToPolarAnglesExp);
NodeFactory.AddNodeAsPrototype('Vision/Geometric and Coordinate Transformations/F_VN_ConvertCartesianToPolarImages', node_F_VN_ConvertCartesianToPolarImages);
NodeFactory.AddNodeAsPrototype('Vision/Geometric and Coordinate Transformations/F_VN_ConvertCartesianToPolarImagesExp', node_F_VN_ConvertCartesianToPolarImagesExp);
NodeFactory.AddNodeAsPrototype('Vision/Geometric and Coordinate Transformations/F_VN_ConvertCartesianToPolarMagnitudeImage', node_F_VN_ConvertCartesianToPolarMagnitudeImage);
NodeFactory.AddNodeAsPrototype('Vision/Geometric and Coordinate Transformations/F_VN_ConvertCartesianToPolarMagnitudes', node_F_VN_ConvertCartesianToPolarMagnitudes);
NodeFactory.AddNodeAsPrototype('Vision/Geometric and Coordinate Transformations/F_VN_ConvertCartesianToPolarPoints', node_F_VN_ConvertCartesianToPolarPoints);
NodeFactory.AddNodeAsPrototype('Vision/Geometric and Coordinate Transformations/F_VN_ConvertCartesianToPolarPointsExp', node_F_VN_ConvertCartesianToPolarPointsExp);
NodeFactory.AddNodeAsPrototype('Vision/Geometric and Coordinate Transformations/F_VN_ConvertPolarToCartesianImages', node_F_VN_ConvertPolarToCartesianImages);
NodeFactory.AddNodeAsPrototype('Vision/Geometric and Coordinate Transformations/F_VN_ConvertPolarToCartesianImagesExp', node_F_VN_ConvertPolarToCartesianImagesExp);
NodeFactory.AddNodeAsPrototype('Vision/Geometric and Coordinate Transformations/F_VN_ConvertPolarToCartesianPoints', node_F_VN_ConvertPolarToCartesianPoints);
NodeFactory.AddNodeAsPrototype('Vision/Geometric and Coordinate Transformations/F_VN_ConvertPolarToCartesianPointsExp', node_F_VN_ConvertPolarToCartesianPointsExp);
NodeFactory.AddNodeAsPrototype('Vision/Geometric and Coordinate Transformations/F_VN_DecomposeAffineTransformation', node_F_VN_DecomposeAffineTransformation);
NodeFactory.AddNodeAsPrototype('Vision/Geometric and Coordinate Transformations/F_VN_DecomposeAffineTransformationExp', node_F_VN_DecomposeAffineTransformationExp);
NodeFactory.AddNodeAsPrototype('Vision/Geometric and Coordinate Transformations/F_VN_DecomposeHomography', node_F_VN_DecomposeHomography);
NodeFactory.AddNodeAsPrototype('Vision/Geometric and Coordinate Transformations/F_VN_DecomposeHomographyExp', node_F_VN_DecomposeHomographyExp);
NodeFactory.AddNodeAsPrototype('Vision/Geometric and Coordinate Transformations/F_VN_FlipImage', node_F_VN_FlipImage);
NodeFactory.AddNodeAsPrototype('Vision/Geometric and Coordinate Transformations/F_VN_GenerateAffineTransformationUnitMatrix2D', node_F_VN_GenerateAffineTransformationUnitMatrix2D);
NodeFactory.AddNodeAsPrototype('Vision/Geometric and Coordinate Transformations/F_VN_GetAffineTransformation', node_F_VN_GetAffineTransformation);
NodeFactory.AddNodeAsPrototype('Vision/Geometric and Coordinate Transformations/F_VN_GetAffineTransformation2D', node_F_VN_GetAffineTransformation2D);
//NodeFactory.AddNodeAsPrototype('Vision/Geometric and Coordinate Transformations/F_VN_GetAffineTransformation2DExp', node_F_VN_GetAffineTransformation2DExp);
NodeFactory.AddNodeAsPrototype('Vision/Geometric and Coordinate Transformations/F_VN_GetPerspectiveTransformation', node_F_VN_GetPerspectiveTransformation);
NodeFactory.AddNodeAsPrototype('Vision/Geometric and Coordinate Transformations/F_VN_Homography', node_F_VN_Homography);
NodeFactory.AddNodeAsPrototype('Vision/Geometric and Coordinate Transformations/F_VN_HomographyExp', node_F_VN_HomographyExp);
NodeFactory.AddNodeAsPrototype('Vision/Geometric and Coordinate Transformations/F_VN_InvertAffineTransformation', node_F_VN_InvertAffineTransformation);
NodeFactory.AddNodeAsPrototype('Vision/Geometric and Coordinate Transformations/F_VN_PerspectiveTransformation', node_F_VN_PerspectiveTransformation);
NodeFactory.AddNodeAsPrototype('Vision/Geometric and Coordinate Transformations/F_VN_PyramidDown', node_F_VN_PyramidDown);
NodeFactory.AddNodeAsPrototype('Vision/Geometric and Coordinate Transformations/F_VN_PyramidUp', node_F_VN_PyramidUp);
NodeFactory.AddNodeAsPrototype('Vision/Geometric and Coordinate Transformations/F_VN_ConvertMaps', node_F_VN_ConvertMaps);
NodeFactory.AddNodeAsPrototype('Vision/Geometric and Coordinate Transformations/F_VN_RemapImage', node_F_VN_RemapImage);
NodeFactory.AddNodeAsPrototype('Vision/Geometric and Coordinate Transformations/F_VN_RemapImageExp', node_F_VN_RemapImageExp);
NodeFactory.AddNodeAsPrototype('Vision/Geometric and Coordinate Transformations/F_VN_RemapImageToLogPolarSpace', node_F_VN_RemapImageToLogPolarSpace);
NodeFactory.AddNodeAsPrototype('Vision/Geometric and Coordinate Transformations/F_VN_RemapImageToLogPolarSpaceExp', node_F_VN_RemapImageToLogPolarSpaceExp);
NodeFactory.AddNodeAsPrototype('Vision/Geometric and Coordinate Transformations/F_VN_RemapImageToLogPolarSpaceExp2', node_F_VN_RemapImageToLogPolarSpaceExp2);
NodeFactory.AddNodeAsPrototype('Vision/Geometric and Coordinate Transformations/F_VN_RemapImageToPolarSpace', node_F_VN_RemapImageToPolarSpace);
NodeFactory.AddNodeAsPrototype('Vision/Geometric and Coordinate Transformations/F_VN_RemapImageToPolarSpaceExp', node_F_VN_RemapImageToPolarSpaceExp);
NodeFactory.AddNodeAsPrototype('Vision/Geometric and Coordinate Transformations/F_VN_RemapImageToPolarSpaceExp2', node_F_VN_RemapImageToPolarSpaceExp2);
NodeFactory.AddNodeAsPrototype('Vision/Geometric and Coordinate Transformations/F_VN_ResizeImage', node_F_VN_ResizeImage);
NodeFactory.AddNodeAsPrototype('Vision/Geometric and Coordinate Transformations/F_VN_ResizeImageExp', node_F_VN_ResizeImageExp);
NodeFactory.AddNodeAsPrototype('Vision/Geometric and Coordinate Transformations/F_VN_ResizeRegion_TcVnRectangle_DINT', node_F_VN_ResizeRegion_TcVnRectangle_DINT);
NodeFactory.AddNodeAsPrototype('Vision/Geometric and Coordinate Transformations/F_VN_RotateImage', node_F_VN_RotateImage);
NodeFactory.AddNodeAsPrototype('Vision/Geometric and Coordinate Transformations/F_VN_RotateImageExp', node_F_VN_RotateImageExp);
NodeFactory.AddNodeAsPrototype('Vision/Geometric and Coordinate Transformations/F_VN_RotateImageExp2', node_F_VN_RotateImageExp2);
NodeFactory.AddNodeAsPrototype('Vision/Geometric and Coordinate Transformations/F_VN_WarpAffine', node_F_VN_WarpAffine);
NodeFactory.AddNodeAsPrototype('Vision/Geometric and Coordinate Transformations/F_VN_WarpAffine_Container', node_F_VN_WarpAffine_Container);
NodeFactory.AddNodeAsPrototype('Vision/Geometric and Coordinate Transformations/F_VN_WarpAffine_Point', node_F_VN_WarpAffine_Point);
NodeFactory.AddNodeAsPrototype('Vision/Geometric and Coordinate Transformations/F_VN_WarpAffine_Rectangle', node_F_VN_WarpAffine_Rectangle);
NodeFactory.AddNodeAsPrototype('Vision/Geometric and Coordinate Transformations/F_VN_WarpAffineExp', node_F_VN_WarpAffineExp);
NodeFactory.AddNodeAsPrototype('Vision/Geometric and Coordinate Transformations/F_VN_WarpPerspective', node_F_VN_WarpPerspective);
NodeFactory.AddNodeAsPrototype('Vision/Geometric and Coordinate Transformations/F_VN_WarpPerspective_Container', node_F_VN_WarpPerspective_Container);
NodeFactory.AddNodeAsPrototype('Vision/Geometric and Coordinate Transformations/F_VN_WarpPerspective_Point', node_F_VN_WarpPerspective_Point);
NodeFactory.AddNodeAsPrototype('Vision/Geometric and Coordinate Transformations/F_VN_WarpPerspective_Rectangle', node_F_VN_WarpPerspective_Rectangle);
NodeFactory.AddNodeAsPrototype('Vision/Geometric and Coordinate Transformations/F_VN_WarpPerspectiveExp', node_F_VN_WarpPerspectiveExp);

// Helpers
NodeFactory.AddNodeAsPrototype('Vision/Helpers/Mux10Way_ITcVnImage', node_Mux10Way_ITcVnImage);

// Image Analysis
//NodeFactory.AddNodeAsPrototype('Vision/Image Analysis/Object Detection/F_VN_AdjustActiveContour', node_F_VN_AdjustActiveContour);
NodeFactory.AddNodeAsPrototype('Vision/Image Analysis/Object Detection/F_VN_SalientFeatures', node_F_VN_SalientFeatures);
NodeFactory.AddNodeAsPrototype('Vision/Image Analysis/Object Detection/F_VN_FindRois', node_F_VN_FindRois);
NodeFactory.AddNodeAsPrototype('Vision/Image Analysis/Object Detection/F_VN_MergeRegions', node_F_VN_MergeRegions);
NodeFactory.AddNodeAsPrototype('Vision/Image Analysis/Object Detection/F_VN_DetectBlobs', node_F_VN_DetectBlobs);
NodeFactory.AddNodeAsPrototype('Vision/Image Analysis/Object Detection/F_VN_DetectBlobsExp', node_F_VN_DetectBlobsExp);
NodeFactory.AddNodeAsPrototype('Vision/Image Analysis/Object Detection/F_VN_FindContourHierarchyExp', node_F_VN_FindContourHierarchyExp);
NodeFactory.AddNodeAsPrototype('Vision/Image Analysis/Object Detection/F_VN_FindContours', node_F_VN_FindContours);
NodeFactory.AddNodeAsPrototype('Vision/Image Analysis/Object Detection/F_VN_FindContoursExp', node_F_VN_FindContoursExp);
NodeFactory.AddNodeAsPrototype('Vision/Image Analysis/Object Detection/F_VN_FindTemplateWalsh', node_F_VN_FindTemplateWalsh);
NodeFactory.AddNodeAsPrototype('Vision/Image Analysis/Object Detection/F_VN_FindTemplateWalsh_AngleRange', node_F_VN_FindTemplateWalsh_AngleRange);
NodeFactory.AddNodeAsPrototype('Vision/Image Analysis/Object Detection/F_VN_FindTemplateWalshExp', node_F_VN_FindTemplateWalshExp);
NodeFactory.AddNodeAsPrototype('Vision/Image Analysis/Object Detection/F_VN_FindTemplateWalshExp_AngleRange', node_F_VN_FindTemplateWalshExp_AngleRange);
NodeFactory.AddNodeAsPrototype('Vision/Image Analysis/Object Detection/F_VN_HoughCircles', node_F_VN_HoughCircles);
NodeFactory.AddNodeAsPrototype('Vision/Image Analysis/Object Detection/F_VN_HoughCirclesExp', node_F_VN_HoughCirclesExp);
NodeFactory.AddNodeAsPrototype('Vision/Image Analysis/Object Detection/F_VN_HoughLines', node_F_VN_HoughLines);
//NodeFactory.AddNodeAsPrototype('Vision/Image Analysis/Object Detection/F_VN_HoughLinesExp', node_F_VN_HoughLinesExp);
NodeFactory.AddNodeAsPrototype('Vision/Image Analysis/Object Detection/F_VN_HoughLinesP', node_F_VN_HoughLinesP);
NodeFactory.AddNodeAsPrototype('Vision/Image Analysis/Object Detection/F_VN_HoughLinesPExp', node_F_VN_HoughLinesPExp);
NodeFactory.AddNodeAsPrototype('Vision/Image Analysis/Object Detection/F_VN_MatchImageHuMoments', node_F_VN_MatchImageHuMoments);
NodeFactory.AddNodeAsPrototype('Vision/Image Analysis/Object Detection/F_VN_MatchTemplate', node_F_VN_MatchTemplate);
NodeFactory.AddNodeAsPrototype('Vision/Image Analysis/Object Detection/F_VN_MatchTemplateAndEvaluate', node_F_VN_MatchTemplateAndEvaluate);
NodeFactory.AddNodeAsPrototype('Vision/Image Analysis/Object Detection/F_VN_MatchTemplateWalsh', node_F_VN_MatchTemplateWalsh);
NodeFactory.AddNodeAsPrototype('Vision/Image Analysis/Object Detection/F_VN_MatchTemplateWalshExp', node_F_VN_MatchTemplateWalshExp);
NodeFactory.AddNodeAsPrototype('Vision/Image Analysis/Object Detection/F_VN_MatchTemplateAndEvaluateExp', node_F_VN_MatchTemplateAndEvaluateExp);
NodeFactory.AddNodeAsPrototype('Vision/Image Analysis/Object Detection/F_VN_MatchTemplateExp', node_F_VN_MatchTemplateExp);
NodeFactory.AddNodeAsPrototype('Vision/Image Analysis/F_VN_CannyEdgeDetection', node_F_VN_CannyEdgeDetection);
NodeFactory.AddNodeAsPrototype('Vision/Image Analysis/F_VN_CannyEdgeDetectionExp', node_F_VN_CannyEdgeDetectionExp);
NodeFactory.AddNodeAsPrototype('Vision/Image Analysis/F_VN_ConnectedComponents', node_F_VN_ConnectedComponents);
NodeFactory.AddNodeAsPrototype('Vision/Image Analysis/F_VN_ConnectedComponentsExp', node_F_VN_ConnectedComponentsExp);
NodeFactory.AddNodeAsPrototype('Vision/Image Analysis/F_VN_ConnectedComponentsWithStats', node_F_VN_ConnectedComponentsWithStats);
NodeFactory.AddNodeAsPrototype('Vision/Image Analysis/F_VN_ConnectedComponentsWithStatsExp', node_F_VN_ConnectedComponentsWithStatsExp);
NodeFactory.AddNodeAsPrototype('Vision/Image Analysis/F_VN_CountNonZeroPixels', node_F_VN_CountNonZeroPixels);
NodeFactory.AddNodeAsPrototype('Vision/Image Analysis/F_VN_DistanceTransformation', node_F_VN_DistanceTransformation);
NodeFactory.AddNodeAsPrototype('Vision/Image Analysis/F_VN_DistanceTransformationExp', node_F_VN_DistanceTransformationExp);
NodeFactory.AddNodeAsPrototype('Vision/Image Analysis/F_VN_GetConnectedComponent', node_F_VN_GetConnectedComponent);
NodeFactory.AddNodeAsPrototype('Vision/Image Analysis/F_VN_GetConnectedComponentExp', node_F_VN_GetConnectedComponentExp);
NodeFactory.AddNodeAsPrototype('Vision/Image Analysis/F_VN_ImageAverage', node_F_VN_ImageAverage);
NodeFactory.AddNodeAsPrototype('Vision/Image Analysis/F_VN_ImageAverageExp', node_F_VN_ImageAverageExp);
NodeFactory.AddNodeAsPrototype('Vision/Image Analysis/F_VN_ImageAverageStdDev', node_F_VN_ImageAverageStdDev);
NodeFactory.AddNodeAsPrototype('Vision/Image Analysis/F_VN_ImageAverageStdDevExp', node_F_VN_ImageAverageStdDevExp);
NodeFactory.AddNodeAsPrototype('Vision/Image Analysis/F_VN_ImageCenterOfMass', node_F_VN_ImageCenterOfMass);
NodeFactory.AddNodeAsPrototype('Vision/Image Analysis/F_VN_ImageCenterOfMassExp', node_F_VN_ImageCenterOfMassExp);
NodeFactory.AddNodeAsPrototype('Vision/Image Analysis/F_VN_ImageMedian', node_F_VN_ImageMedian);
NodeFactory.AddNodeAsPrototype('Vision/Image Analysis/F_VN_ImageMedianExp', node_F_VN_ImageMedianExp);
NodeFactory.AddNodeAsPrototype('Vision/Image Analysis/F_VN_ImageMoments', node_F_VN_ImageMoments);
NodeFactory.AddNodeAsPrototype('Vision/Image Analysis/F_VN_MaxPixelValue', node_F_VN_MaxPixelValue);
NodeFactory.AddNodeAsPrototype('Vision/Image Analysis/F_VN_MaxPixelValueExp', node_F_VN_MaxPixelValueExp);
NodeFactory.AddNodeAsPrototype('Vision/Image Analysis/F_VN_MinPixelValue', node_F_VN_MinPixelValue);
NodeFactory.AddNodeAsPrototype('Vision/Image Analysis/F_VN_MinPixelValueExp', node_F_VN_MinPixelValueExp);
NodeFactory.AddNodeAsPrototype('Vision/Image Analysis/F_VN_RegionOrientation', node_F_VN_RegionOrientation);
NodeFactory.AddNodeAsPrototype('Vision/Image Analysis/F_VN_RegionOrientationExp', node_F_VN_RegionOrientationExp);
NodeFactory.AddNodeAsPrototype('Vision/Image Analysis/F_VN_ImageAbsoluteAverage', node_F_VN_ImageAbsoluteAverage);
NodeFactory.AddNodeAsPrototype('Vision/Image Analysis/F_VN_UprightInnerRectangle', node_F_VN_UprightInnerRectangle);
NodeFactory.AddNodeAsPrototype('Vision/Image Analysis/F_VN_UprightInnerRectangleExp', node_F_VN_UprightInnerRectangleExp);

// Image Color and Contrast Processing
NodeFactory.AddNodeAsPrototype('Vision/Image Color and Contrast Processing/F_VN_ApplyColorMap', node_F_VN_ApplyColorMap);
//NodeFactory.AddNodeAsPrototype('Vision/Image Color and Contrast Processing/F_VN_ApplyLut', node_F_VN_ApplyLut);
NodeFactory.AddNodeAsPrototype('Vision/Image Color and Contrast Processing/F_VN_Clahe', node_F_VN_Clahe);
NodeFactory.AddNodeAsPrototype('Vision/Image Color and Contrast Processing/F_VN_ClaheExp', node_F_VN_ClaheExp);
NodeFactory.AddNodeAsPrototype('Vision/Image Color and Contrast Processing/F_VN_ConvertColorSpace', node_F_VN_ConvertColorSpace);
NodeFactory.AddNodeAsPrototype('Vision/Image Color and Contrast Processing/F_VN_GenerateColorMap', node_F_VN_GenerateColorMap);
NodeFactory.AddNodeAsPrototype('Vision/Image Color and Contrast Processing/F_VN_GenerateCustomColorMap', node_F_VN_GenerateCustomColorMap);
NodeFactory.AddNodeAsPrototype('Vision/Image Color and Contrast Processing/F_VN_Histogram', node_F_VN_Histogram);
NodeFactory.AddNodeAsPrototype('Vision/Image Color and Contrast Processing/F_VN_HistogramEqualization', node_F_VN_HistogramEqualization);
NodeFactory.AddNodeAsPrototype('Vision/Image Color and Contrast Processing/F_VN_HistogramEqualizationExp', node_F_VN_HistogramEqualizationExp);
NodeFactory.AddNodeAsPrototype('Vision/Image Color and Contrast Processing/F_VN_HistogramExp', node_F_VN_HistogramExp);
NodeFactory.AddNodeAsPrototype('Vision/Image Color and Contrast Processing/F_VN_InvertImageColor', node_F_VN_InvertImageColor);
NodeFactory.AddNodeAsPrototype('Vision/Image Color and Contrast Processing/F_VN_InvertImageColorExp', node_F_VN_InvertImageColorExp);
NodeFactory.AddNodeAsPrototype('Vision/Image Color and Contrast Processing/F_VN_NormalizeImage', node_F_VN_NormalizeImage);
NodeFactory.AddNodeAsPrototype('Vision/Image Color and Contrast Processing/F_VN_NormalizeImageExp', node_F_VN_NormalizeImageExp);
NodeFactory.AddNodeAsPrototype('Vision/Image Color and Contrast Processing/F_VN_NormalizeImageForDisplay', node_F_VN_NormalizeImageForDisplay);
//NodeFactory.AddNodeAsPrototype('Vision/Image Color and Contrast Processing/F_VN_ReferenceColorSimilarity_ITcVnColorModel', node_F_VN_ReferenceColorSimilarity_ITcVnColorModel);
//NodeFactory.AddNodeAsPrototype('Vision/Image Color and Contrast Processing/F_VN_ReferenceColorSimilarity_ITcVnMlModel', node_F_VN_ReferenceColorSimilarity_ITcVnMlModel);
NodeFactory.AddNodeAsPrototype('Vision/Image Color and Contrast Processing/F_VN_ReferenceColorSimilarity_TcVnVector3_LREAL', node_F_VN_ReferenceColorSimilarity_TcVnVector3_LREAL);
//NodeFactory.AddNodeAsPrototype('Vision/Image Color and Contrast Processing/F_VN_ReferenceColorSimilarityExp_ITcVnColorModel', node_F_VN_ReferenceColorSimilarityExp_ITcVnColorModel);
//NodeFactory.AddNodeAsPrototype('Vision/Image Color and Contrast Processing/F_VN_ReferenceColorSimilarityExp_ITcVnMlModel', node_F_VN_ReferenceColorSimilarityExp_ITcVnMlModel);
NodeFactory.AddNodeAsPrototype('Vision/Image Color and Contrast Processing/F_VN_ReferenceColorSimilarityExp_TcVnVector3_LREAL', node_F_VN_ReferenceColorSimilarityExp_TcVnVector3_LREAL);
//NodeFactory.AddNodeAsPrototype('Vision/Image Color and Contrast Processing/F_VN_TrainImageColor', node_F_VN_TrainImageColor);
//NodeFactory.AddNodeAsPrototype('Vision/Image Color and Contrast Processing/F_VN_TrainImageColor_ITcVnMlModel', node_F_VN_TrainImageColor_ITcVnMlModel);
//NodeFactory.AddNodeAsPrototype('Vision/Image Color and Contrast Processing/F_VN_TrainImageColorExp', node_F_VN_TrainImageColorExp);
//NodeFactory.AddNodeAsPrototype('Vision/Image Color and Contrast Processing/F_VN_TrainImageColorExp_ITcVnMlModel', node_F_VN_TrainImageColorExp_ITcVnMlModel);
//NodeFactory.AddNodeAsPrototype('Vision/Image Color and Contrast Processing/F_VN_TrainImageColorExp2', node_F_VN_TrainImageColorExp2);
//NodeFactory.AddNodeAsPrototype('Vision/Image Color and Contrast Processing/F_VN_TrainImageColorExp2_ITcVnMlModel', node_F_VN_TrainImageColorExp2_ITcVnMlModel);
NodeFactory.AddNodeAsPrototype('Vision/Image Color and Contrast Processing/F_VN_WhiteBalance', node_F_VN_WhiteBalance);

